# B&R Automation Studio project ComauRacer3demo (part 2)

### Config_3.mechanicalsystem - X20CP1586/mappMotion/6AxesRoboArmA/Config_3.mechanicalsystem
```
Element MechSys_6AxRobA (Type=mechanicalsystem)
  Type = 6AxesRoboarm
    Subtype = 6AxesRoboarmA
      Description = Standard
        Dimensions:
          TranslationFromBaseToQ1IsReadOnly = 0
          TranslationFromBaseToQ1:
            X = 0.0
            Y = 0.0
            Z = 0.0
          TranslationFromQ1ToQ2IsReadOnly = 0
          TranslationFromQ1ToQ2:
            X = 250.0
            Y = 0.0
            Z = 640.0
          TranslationFromQ2ToQ3IsReadOnly = 0
          TranslationFromQ2ToQ3:
            X = 0.0
            Y = 0.0
            Z = 630.0
          TranslationFromQ3ToQ4IsReadOnly = 0
          TranslationFromQ3ToQ4:
            X = 827.5
            Y = 0.0
            Z = 196.0
          TranslationFromQ4ToQ5IsReadOnly = 0
          TranslationFromQ4ToQ5:
            X = 0.0
          TranslationFromQ5ToQ6IsReadOnly = 0
          TranslationFromQ5ToQ6:
            X = 160.0
          TranslationFromQ6ToFlange:
            X = 0.0
            Y = 0.0
            Z = 0.0
        Offsets:
          JointAxisIsReadOnly = 0
          JointAxis[1] = 0.0
          JointAxis[2] = 0.0
          JointAxis[3] = 0.0
          JointAxis[4] = 0.0
          JointAxis[5] = 0.0
          JointAxis[6] = 0.0
        CountDirections:
          JointAxisIsReadOnly = 0
          JointAxis[1] = Standard
          JointAxis[2] = Standard
          JointAxis[3] = Standard
          JointAxis[4] = Standard
          JointAxis[5] = Standard
          JointAxis[6] = Standard
      CoordinatesNames = Default
        XCoordinateName = X
        YCoordinateName = Y
        ZCoordinateName = Z
        ACoordinateName = A
        BCoordinateName = B
        CCoordinateName = C
      WireFrameModel = Standard
        Q1ToQ2 = ConnectionLine
          Distance = 0.0
        Q2ToQ3 = ConnectionLine
          Distance = 0.0
        Q3ToQ4 = ConnectionLine
          Distance = 0.0
        Q4ToQ5 = ConnectionLine
          Distance = 0.0
        Q5ToQ6 = ConnectionLine
          Distance = 0.0
        Q6ToFlange = ConnectionLine
          Distance = 0.0
        FlangeToTcp = ConnectionLine
          Distance = 0.0
      DynamicModel = DynParTable
        TableRef
      InternalDynamicModel = NotUsed
      JointAxesPositionLimits:
        JointAxis[1] = UseAxisLimits
        JointAxis[2] = UseAxisLimits
        JointAxis[3] = UseAxisLimits
        JointAxis[4] = UseAxisLimits
        JointAxis[5] = UseAxisLimits
        JointAxis[6] = UseAxisLimits
```

## Logical view

Binary libraries used (declarations not repeated): operator, runtime, astime, AsIecCon, MpRobotics, McAxGroup, MpBase, McBase, CoTrace, AsZip, FileIO, sys_lib, McAcpAx, McAxis, MpAxis, McAcpPar, McPathGen, McProgInt, MpAudit 5.14.1, MpServer, MpAlarmX 5.14.1, MpUserX 5.14.1, MpFile 5.14.1, AsBrStr, MpRecipe 5.14.1

### Global.typ - Global data types
```iecst
TYPE
	R3ManualModeType : 	STRUCT  (*Manual mode type*)
		AxisButton : R3TCPAxisBtnType; (*Stores button states for global coordinate system*)
		JointButton : R3JointBtnType; (*Stores button states for axis coordinate system*)
		Velocity : REAL; (*Stores set velocity*)
		Acceleration : REAL; (*Stores set acceleration*)
		Deceleration : REAL; (*Stores set deceleration*)
		CoordinateSystem : UDINT; (*Stores selected coordinate system (0 - axis, 9 - global, 10 - tool) (no tool is set, so 9=10)*)
		Direction : DirectionEnum; (*Stores which direction should the axis be moved*)
	END_STRUCT;
	R3JointBtnType : 	STRUCT  (*Axes 1-6 select button*)
		Q1 : BOOL;
		Q2 : BOOL;
		Q3 : BOOL;
		Q4 : BOOL;
		Q5 : BOOL;
		Q6 : BOOL;
	END_STRUCT;
	R3TCPAxisBtnType : 	STRUCT  (*Global Coordinate System Select button*)
		X : BOOL;
		Y : BOOL;
		Z : BOOL;
		A : BOOL;
		B : BOOL;
		C : BOOL;
	END_STRUCT;
	DirectionEnum :
		(
		POSITIVE,
		NEGATIVE
		);
END_TYPE
```

### Global.var - Global variables
```iecst
VAR RETAIN
	gIsCalibrated : BOOL;
	gRacer3HomeRestorePos : ARRAY[0..5] OF McAcpAxRestorePosType; (*Permanent - stores home position, set in calibration process*)
	gRacer3ZeroPosition : ARRAY[0..5] OF LREAL; (*Position of axes saved after calibration*)
END_VAR
VAR
	gActiveContent : INT := 1;
END_VAR
```

### Package Logical/Libraries - Global libraries

### Library Logical/Libraries/RacerLib (IEC)

#### Types.typ - Exported data types
```iecst
TYPE
	R3AutomaticModeErrorEnum :
		(
		autoNO_ERROR := 0,
		autoLOAD_PROGRAM_ERROR := 1,
		autoUNLOAD_PROGRAM_ERROR := 2,
		autoEXECUTE_PROGRAM_ERROR := 3,
		autoPAUSE_ERROR := 4,
		autoCONTINUE_ERROR := 5,
		autoABORT_ERROR := 6
		);
	R3AutomaticModeCmds : 	STRUCT  (*Automatic mode commands*)
		LoadProgram : MC_BR_LoadProgram;
		ExecuteProgram : MC_BR_MoveProgram;
		UnloadProgram : MC_BR_UnloadProgram;
		PauseProgram : MC_GroupInterrupt;
		ContinueProgram : MC_GroupContinue;
		GroupStop : MC_GroupStop;
	END_STRUCT;
	R3AutomaticModeState :
		( (*Automatic mode state machine*)
		autoSTATE_WAIT := 1, (*waiting for instruction*)
		autoSTATE_LOAD := 2, (*loading program*)
		autoSTATE_UNLOAD := 3, (*Unloading program state*)
		autoSTATE_EXECUTE := 4, (*executing program*)
		autoSTATE_DONE := 5, (*execution done*)
		autoSTATE_PAUSE := 6, (*program paused*)
		autoSTATE_CONTINUE := 7, (*Continues paused program*)
		autoSTATE_ABORT := 8, (*Abort current program*)
		autoSTATE_ERROR := 0 (*error state*)
		);
	R3AutomaticModePara : 	STRUCT  (*Automatic mode parameters*)
		ProgramName : STRING[260]; (*Program name to load/execute*)
		Load : BOOL; (*Load a program*)
		Execute : BOOL; (*Executes a program*)
		Unload : BOOL; (*Unloads a program*)
		ErrorReset : BOOL; (*Resets errors*)
		Abort : BOOL; (*Aborts execution.*)
		UnloadAll : BOOL; (*tells the program to unload all programs from memory (used with Unload)*)
		Pause : BOOL; (*Pauses execution*)
		Continue : BOOL; (*Continues execution*)
		Continuous : BOOL; (*Defines whether the program will be called continuously*)
	END_STRUCT;
	R3AutomaticModeInfo : 	STRUCT
		CurrentState : R3AutomaticModeState; (*Current automode state*)
		Error : R3AutomaticModeErrorEnum;
		ErrorID : DINT;
		Paused : BOOL;
		IsError : BOOL; (*Only for visualisation.*)
	END_STRUCT;
	R3AutomaticModeType : 	STRUCT  (*Automatic mode main structure*)
		Parameters : R3AutomaticModePara;
		Info : R3AutomaticModeInfo;
		Cmds : R3AutomaticModeCmds;
	END_STRUCT;
	R3WorkspaceType : 	STRUCT  (*this allows workspace to be set during runtime.*)
		Para : McCfgAxGrpFeatWsmType := (ModalDataBehaviour:=(Type:=mcAGFMDB_USE_AX_GRP_SET));
		Cmd : MC_BR_ProcessConfig;
		Done : BOOL; (*indicates the FB has finished*)
	END_STRUCT;
	R3ManualModeType : 	STRUCT  (*Manual mode type*)
		AxisButton : R3AxisBtnType; (*Stores button states for select coordinate system*)
		CoordinateSystem : McCoordinateSystemEnum; (*Stores selected coordinate system (0 - axis, 9 - global, 10 - tool) (no tool is set, so 9=10)*)
		Direction : INT; (*Stores which direction should the axis be moved (1 - POSITIVE, -1 - NEGATIVE)*)
		JogVelocity : REAL := 20; (*Stores the velocity of axis*)
		PathLimits : McJogPathLimitsType; (*Stores set limits of acceleration and deceleration, velocity and jerk*)
		ActivateMove : BOOL; (*Enables or disables current move execution*)
		ExitManual : BOOL; (*Exits Manual Mode on True*)
	END_STRUCT;
	R3AxisBtnType : 	STRUCT  (*Global Coordinate System Select button*)
		Q1 : BOOL;
		Q2 : BOOL;
		Q3 : BOOL;
		Q4 : BOOL;
		Q5 : BOOL;
		Q6 : BOOL;
	END_STRUCT;
	R3DirectionEnum :
		( (*Currently unused*)
		POSITIVE := 1,
		NEGATIVE := -1
		);
	R3StateMachineEnum :
		(
		STATE_ERROR, (*Error state*)
		STATE_INIT, (*Initialisation state*)
		STATE_POWER_ON, (*Powering on state*)
		STATE_READY, (*Ready for commands*)
		STATE_MANUAL_CONTROL, (*Manual mode*)
		STATE_SEMI_AUTOMATIC, (*Semi automatic mode*)
		STATE_AUTOMATIC, (*Automatic mode (script execution)*)
		STATE_CALIBRATION, (*Calibration mode*)
		STATE_HOMING, (*Homing mode*)
		STATE_BRAKES (*This will read brakes' status.*)
		);
	R3CalibrationType : 	STRUCT
		CalibrationState : R3CalibrationStateEnum; (*State machine used to control Calibration behaviour*)
		CalibrationModePara : R3ManualModeType; (*same type used for manual mode (slightly different code handling)*)
		AxisCalibrated : ARRAY[0..5]OF BOOL := [6(0)]; (*Saves which axes have been calibrated (defaults to 0 upon creation)*)
		AxisSaveBtn : BOOL; (*Button to save current position as calibrated*)
		Axis5To6Para : R3Axis5To6Type; (*Stores axis 4 and 5 settings for axis 5 and 6 calibration*)
		SavedPositions : ARRAY[0..5]OF LREAL;
		InitHome : MC_BR_InitHome_AcpAx; (*Used to init home positions after each save*)
		InitHomePara : McAcpAxHomingParType; (*Homing parameters after each save*)
		AxesRef : ARRAY[0..5]OF UDINT; (*Axes reference.*)
	END_STRUCT;
	R3CalibrationStateEnum :
		(
		STATE_START,
		STATE_CALIBRATE_Q1,
		STATE_CALIBRATE_Q2,
		STATE_CALIBRATE_Q3,
		STATE_CALIBRATE_Q4,
		STATE_CALIBRATE_Q5,
		STATE_CALIBRATE_Q6,
		STATE_RESTORE_Q3_Q5
		);
	R3Axis5To6Type : 	STRUCT  (*Type for storing axis 3 and 5 settings for axes 5 and 6 calibration*)
		Axis3Moved : BOOL; (*Stores whether axis 3 has been moved in order to calibrate axes 5 and  6*)
		Axis5Moved : BOOL; (*Stores whether axis 5 has been moved in order to calibrate axis 6*)
		AxisMoveVelocity : REAL; (*Velocity of axis 3 and 5*)
		Axis3Angle : LREAL := -45.0; (*Angle of axis 3 to be set*)
		Axis5Angle : LREAL := -118.0; (*Angle of axis 5 to be set*)
		Axis5Return : BOOL; (*Flag to be set by a button to restore axis 3 and 5's positions after calibrating axis 6*)
		Axis35Restored : BOOL; (*Axis 3 and 5 have been restored to previous position*)
	END_STRUCT;
	R3SemiAutoEnumType :
		(
		INIT := 0,
		START := 1,
		UPDATE := 2,
		GO := 3,
		STATE_STOP := 5,
		STATE_PAUSE := 4
		);
	R3SemiAutoModeType : 	STRUCT
		AskedValue : R3AskedValueType; (*Stores given axis distance for relative move*)
		Flag : BOOL; (*Flag between READY and SEMIAUTO*)
		Mode : BOOL; (*Switches between relative and absolute modes, 1 for Relative, 0 for Absolute*)
		UpdatePending : BOOL; (*if UpdatePending then updates before starting move*)
		State : R3SemiAutoEnumType; (*state selector for state machine*)
		ModeForThisMove : BOOL; (*makes sure that switching mode in time of moving doesnt bugs out move*)
		CoordinateSystem : McCoordinateSystemEnum; (*Stores selected coordinate system (0 - axis, 9 - global, 10 - tool) (no tool is set, so 9=10)*)
		PathMode : BOOL; (*Switches between direct and linear path mode, 1 for linear , 0 for direct*)
		PathModeForThisMove : BOOL;
		ExitSemiAuto : BOOL;
		Pause : BOOL;
	END_STRUCT;
	ControlSelectEnum :
		(
		ManualJog := 1,
		SemiAutomatic := 2,
		Automatic := 3,
		None := 0
		);
	R3AskedValueType : 	STRUCT  (*for SemiAuto*)
		Velocity : REAL := 69;
		Acceleration : REAL := 100;
		Deceleration : REAL := 100;
		Jerk : REAL := 0;
		TCS : ARRAY[0..5]OF REAL := [420,420,420,69,69,69];
		ACS : ARRAY[0..5]OF REAL := [-69,69,69,69,-69,69];
	END_STRUCT;
	R3CalibrationMainType : 	STRUCT
		Info : CalibrationInfo; (*Information portion of calibration.*)
		Cmds : CalibrationCmds; (*Calibration commands*)
		Para : CalibrationParaType; (*Calibration parameters*)
	END_STRUCT;
	CalibrationParaType : 	STRUCT
		Parameters : R3CalibrationType;
		HomingParameters : McAcpAxHomingParType;
		FakeHomingModeEnum : ARRAY[0..14]OF McHomingModeEnum := [15(mcHOMING_DIRECT)];
		Positions : ARRAY[0..14]OF LREAL := [15(0.0)];
		HomingModeEnum : ARRAY[0..14]OF McHomingModeEnum := [15(mcHOMING_INIT)];
	END_STRUCT;
	CalibrationCmds : 	STRUCT
		Mode : R3CalibrationMode;
		InitHome : MC_BR_InitHome_AcpAx;
		GroupHome : MC_BR_GroupHome_15;
	END_STRUCT;
	CalibrationInfo : 	STRUCT
		CurrentState : OuterCalibrationState;
	END_STRUCT;
	OuterCalibrationState :
		(
		STATE_BEGIN,
		STATE_FAKE_HOME,
		STATE_MOVING,
		STATE_SAVING_POSITION,
		STATE_DONE
		);
	CommunicationType : 	STRUCT
		Power : BOOL := FALSE;
		Pause : BOOL := FALSE;
		Stop : BOOL := FALSE;
		ErrorReset : BOOL := FALSE;
		ModeSystem : BOOL := TRUE;
		PathSystem : BOOL := TRUE;
		changeModePending : USINT := 0; (*1-Manual       2-SemiManual      3-Auto 0-none*)
		NOTPathSystem : BOOL;
		NOTModeSystem : BOOL;
		CoordinateSystemManual : BOOL := FALSE;
		NOTCoordinateSystemSemiAuto : BOOL := FALSE;
		CoordinateSystemSemiAuto : BOOL := FALSE;
		NOTCoordinateSystem : BOOL;
		txt_State_out : WSTRING[80];
		AskedMaxVelocity : REAL; (*not needed*)
		AskedMaxAcc : REAL; (*not needed*)
		AskedMaxDeAcc : REAL; (*not needed*)
		AskedAutoJerk : REAL; (*not needed*)
		AskedAutoDeAcc : REAL; (*not needed*)
		AskedAutoAcc : REAL; (*not needed*)
		AskedAutoVelocity : REAL; (*not needed*)
		AskedManualVelocity : REAL; (*not needed*)
		UpdateSemiAutoVars : BOOL := FALSE;
		CalibBtn1To5 : BOOL := FALSE;
		CalibrationImage : STRING[80];
		TextManager : TextManagerType;
		RestoreAxis5 : BOOL := FALSE;
		CalibrateAgain : BOOL := FALSE;
		txt_State_out_front : STRING[80];
		BrakeOpen : BOOL; (*open the brakes*)
		BrakeClose : BOOL; (*close the brakes*)
		BrakeReadStatus : BOOL; (*read status of brakes*)
		BrakesSet : BOOL; (*This variable tells the program if brake parameters have been set.*)
		ToolOutput : BOOL; (*This variable enables tool control*)
		ReturnToZero : BOOL; (*This variable allows returning to zero position in manual mode.*)
		ResetHome : BOOL;
		WarmRestart : BOOL := FALSE;
		ReadWorkspace : BOOL;
	END_STRUCT;
	R3BrakeStateMachineEnum :
		(
		brakeREAD,
		brakeOPEN,
		brakeCLOSE,
		brakeDONE,
		brakeERROR
		);
	R3BrakeParaType : 	STRUCT
		BrakeCmd : McBrakeCmdEnum;
		Identifier : UDINT;
	END_STRUCT;
	R3BrakeCmdsType : 	STRUCT
		BrakeOperation : MC_BR_GroupBrakeOperation;
	END_STRUCT;
	R3BrakeInfoType : 	STRUCT
		BrakeStatus : ARRAY[1..2]OF McBrakeStatusEnum;
		Done : BOOL;
		State : R3BrakeStateMachineEnum;
		Error : BOOL;
	END_STRUCT;
	R3BrakeType : 	STRUCT
		Parameters : R3BrakeParaType;
		Info : R3BrakeInfoType;
		Cmds : R3BrakeCmdsType;
	END_STRUCT;
	R3KeyCheckType : 	STRUCT
		original_combo : ARRAY[0..4]OF USINT := [1,2,3,0,17];
		pending_combo : ARRAY[0..4]OF USINT;
		i : USINT := 0;
		temp_value : USINT;
		value_changed : BOOL := FALSE;
		event_achieved : BOOL := FALSE;
	END_STRUCT;
	TextManagerType : 	STRUCT
		CalibHelper : STRING[80];
	END_STRUCT;
END_TYPE
```

#### Constants.var - Exported constants
```iecst
VAR CONSTANT
	gAlarmXCore : USINT := 0;
END_VAR
```

#### RacerLib.fun - Exported functions and function blocks
```iecst
FUNCTION_BLOCK R3BrakeSet
	VAR_INPUT
		Axis1 : REFERENCE TO UDINT;
		Axis2 : REFERENCE TO UDINT;
		Axis3 : REFERENCE TO UDINT;
		Axis4 : REFERENCE TO UDINT;
		Axis5 : REFERENCE TO UDINT;
		Axis6 : REFERENCE TO UDINT;
	END_VAR
	VAR_OUTPUT
		Done : BOOL;
		Error : BOOL;
	END_VAR
	VAR
		BrakePara : McAcpAxBrakeParType;
		CurrentAxis : USINT := 1;
		BrakeSet : MC_BR_BrakeSetPar_AcpAx;
	END_VAR
END_FUNCTION_BLOCK

{REDUND_ERROR} FUNCTION_BLOCK R3ManualMode (*TODO: Add your comment here*) (*$GROUP=User,$CAT=User,$GROUPICON=User.png,$CATICON=User.png*)
	VAR_INPUT
		ManualModePara : R3ManualModeType;
	END_VAR
	VAR_IN_OUT
		RoboArm : MpRoboArm6Axis;
		RoboArmPara : MpRoboArm6AxisParType;
		MainState : R3StateMachineEnum;
		ControlSelector : ControlSelectEnum;
	END_VAR
	VAR
		j : USINT;
		JogVelocityActual : REAL;
	END_VAR
END_FUNCTION_BLOCK

{REDUND_ERROR} FUNCTION_BLOCK R3SemiAutoMode (*TODO: Add your comment here*) (*$GROUP=User,$CAT=User,$GROUPICON=User.png,$CATICON=User.png*)
	VAR_IN_OUT
		SemiAutoModePara : R3SemiAutoModeType;
		RoboArm : MpRoboArm6Axis;
		RoboArmPara : MpRoboArm6AxisParType;
		MainState : R3StateMachineEnum;
		ControlSelector : ControlSelectEnum;
	END_VAR
	VAR
		SemiAutoModePara_memory : R3SemiAutoModeType;
		WeNeedToGoBack : BOOL;
		IsPaused : BOOL;
	END_VAR
END_FUNCTION_BLOCK

{REDUND_UNREPLICABLE} FUNCTION_BLOCK R3CalibrationMode
	VAR_IN_OUT
		CalibrationPara : R3CalibrationType;
		RoboArm : MpRoboArm6Axis;
		RoboArmPara : MpRoboArm6AxisParType;
	END_VAR
	VAR
		JogVelocityActual : {REDUND_UNREPLICABLE} REAL;
		j : {REDUND_UNREPLICABLE} USINT;
	END_VAR
END_FUNCTION_BLOCK

{REDUND_ERROR} FUNCTION checkAxisLimits : BOOL (*returns TRUE if semi-automatic path is containted in axis limits, check is for relative positions*) (*$GROUP=User,$CAT=User,$GROUPICON=User.png,$CATICON=User.png*)
	VAR_INPUT
		Q1 : REAL;
		Q2 : REAL;
		Q3 : REAL;
		Q4 : REAL;
		Q5 : REAL;
		Q6 : REAL;
		Mode : BOOL; (*1 for relative, 0 for absolute*)
		RoboArm : MpRoboArm6Axis; (*needed for current axis position*)
	END_VAR
END_FUNCTION

{REDUND_ERROR} {REDUND_UNREPLICABLE} FUNCTION_BLOCK R3AutomaticMode (*TODO: Add your comment here*) (*$GROUP=User,$CAT=User,$GROUPICON=User.png,$CATICON=User.png*)
	VAR_INPUT
		AxesGroup : REFERENCE TO UDINT; (*AxesGroup to execute program on*)
	END_VAR
	VAR_IN_OUT
		AutoMode : R3AutomaticModeType; (*Main type variable*)
	END_VAR
	VAR
		UnloadMode : {REDUND_UNREPLICABLE} McUnloadProgramModeEnum; (*defines unload mode behaviour*)
	END_VAR
END_FUNCTION_BLOCK

{REDUND_ERROR} {REDUND_UNREPLICABLE} FUNCTION_BLOCK R3Workspace (*TODO: Add your comment here*) (*$GROUP=User,$CAT=User,$GROUPICON=User.png,$CATICON=User.png*)
	VAR_IN_OUT
		Para : R3WorkspaceType;
	END_VAR
END_FUNCTION_BLOCK
```

#### R3ManualMode.st
```iecst
(* TODO: Add your comment here *)
FUNCTION_BLOCK R3ManualMode

	IF ManualModePara.Direction = 1 THEN // set actual axis velocity based on which direction it's set to be moved
		JogVelocityActual := ManualModePara.JogVelocity;
	ELSIF ManualModePara.Direction = -1 THEN
		JogVelocityActual := -1 * ManualModePara.JogVelocity;
	ELSIF  ManualModePara.Direction = 0 THEN
		JogVelocityActual := 0;
	END_IF

	RoboArmPara.Jog.CoordSystem := ManualModePara.CoordinateSystem;
	RoboArmPara.Jog.PathLimits := ManualModePara.PathLimits;

	IF ManualModePara.ActivateMove THEN
		(* old Szymon's version
		IF ManualModePara.AxisButton.Q1 THEN // if a button is pressed, write corresponding velocity to the jog velocity array
			//IF RoboArmPara.Jog.Velocity[0] <> JogVelocityActual THEN // test if this fixes strange movement style
				RoboArmPara.Jog.Velocity[0] := JogVelocityActual;
			//END_IF
		ELSIF ManualModePara.AxisButton.Q2 THEN
			//IF RoboArmPara.Jog.Velocity[1] <> JogVelocityActual THEN
				RoboArmPara.Jog.Velocity[1] := JogVelocityActual;
			//END_IF
		ELSIF ManualModePara.AxisButton.Q3 THEN
			RoboArmPara.Jog.Velocity[2] := JogVelocityActual;

		ELSIF ManualModePara.AxisButton.Q4 THEN
			RoboArmPara.Jog.Velocity[3] := JogVelocityActual;

		ELSIF ManualModePara.AxisButton.Q5 THEN
			RoboArmPara.Jog.Velocity[4] := JogVelocityActual;

		ELSIF ManualModePara.AxisButton.Q6 THEN
			RoboArmPara.Jog.Velocity[5] := JogVelocityActual;

		ELSE //if no buttons are pressed reset jog velocity array

			FOR j := 0 TO 5 BY 1 DO //set every jog velocity to 0
				RoboArmPara.Jog.Velocity[j] := 0.0;
			END_FOR;
		END_IF
		*)

		IF ManualModePara.AxisButton.Q1 THEN
			RoboArmPara.Jog.Velocity[0] := JogVelocityActual;
		ELSE
			RoboArmPara.Jog.Velocity[0] := 0;
		END_IF

		IF ManualModePara.AxisButton.Q2 THEN
			RoboArmPara.Jog.Velocity[1] := JogVelocityActual;
		ELSE
			RoboArmPara.Jog.Velocity[1] := 0;
		END_IF

		IF ManualModePara.AxisButton.Q3 THEN
			RoboArmPara.Jog.Velocity[2] := JogVelocityActual;
		ELSE
			RoboArmPara.Jog.Velocity[2] := 0;
		END_IF

		IF ManualModePara.AxisButton.Q4 THEN
			RoboArmPara.Jog.Velocity[3] := JogVelocityActual;
		ELSE
			RoboArmPara.Jog.Velocity[3] := 0;
		END_IF

		IF ManualModePara.AxisButton.Q5 THEN
			RoboArmPara.Jog.Velocity[4] := JogVelocityActual;
		ELSE
			RoboArmPara.Jog.Velocity[4] := 0;
		END_IF

		IF ManualModePara.AxisButton.Q6 THEN
			RoboArmPara.Jog.Velocity[5] := JogVelocityActual;
		ELSE
			RoboArmPara.Jog.Velocity[5] := 0;
		END_IF
		IF RoboArm.Jog <> TRUE THEN
			RoboArm.Jog := TRUE;
		END_IF
	ELSE
		RoboArm.Jog := FALSE;
	END_IF

	IF ManualModePara.ExitManual THEN
		//clean up
		ManualModePara.Direction:=0;
		JogVelocityActual:=0;
		FOR j := 0 TO 5 BY 1 DO //set every jog velocity to 0
				RoboArmPara.Jog.Velocity[j] := 0;
		END_FOR;
		ManualModePara.ActivateMove:=FALSE;
		RoboArm.Jog:=FALSE;
		//go out
		ManualModePara.ExitManual := FALSE;
	END_IF

END_FUNCTION_BLOCK
```

#### R3SemiAutoMode.st
```iecst
FUNCTION_BLOCK R3SemiAutoMode

	IF SemiAutoModePara.ExitSemiAuto THEN
		SemiAutoModePara.State := STATE_STOP;
	END_IF

	(*
	IF SemiAutoModePara.Pause THEN
		SemiAutoModePara_memory := SemiAutoModePara;
		RoboArm.MoveDirect:=FALSE;
		RoboArm.MoveLinear:=FALSE;
		SemiAutoModePara.Flag:=FALSE;
	END_IF
	*)
	CASE SemiAutoModePara.State OF
		INIT:
			IF SemiAutoModePara.UpdatePending THEN
				SemiAutoModePara.State := UPDATE;
			ELSE
				SemiAutoModePara.State := START;
			END_IF

			//TODO CHECK AXIS LIMITS AND SINGULAR POINT AND SEND ERROR (ALARM) AND AVOID MOVING
			//IF checkAxisLimits(Q1:=SemiAutoModePara.AskedValue.Q0,Q2:=SemiAutoModePara.AskedValue.Q1,Q3:=SemiAutoModePara.AskedValue.Q2,Q4:=SemiAutoModePara.AskedValue.Q3,Q5:=SemiAutoModePara.AskedValue.Q4,Q6:=SemiAutoModePara.AskedValue.Q5,Mode := SemiAutoModePara.ModeForThisMove, RoboArm:=RoboArm) THEN
			// send alarm out of bounds
			//MpAlarmXSet(gAlarmXCore, 'OutOfLimits');
			//END_IF

			// check for singular point and send alarm

		UPDATE:

			RoboArmPara.CoordSystem := SemiAutoModePara.CoordinateSystem;

			RoboArmPara.Velocity := SemiAutoModePara.AskedValue.Velocity;
			RoboArmPara.Acceleration := SemiAutoModePara.AskedValue.Acceleration;
			RoboArmPara.Deceleration := SemiAutoModePara.AskedValue.Deceleration;
			RoboArmPara.Jerk := SemiAutoModePara.AskedValue.Jerk;

			SemiAutoModePara.ModeForThisMove:=SemiAutoModePara.Mode;
			SemiAutoModePara.PathModeForThisMove:=SemiAutoModePara.PathMode;

			IF SemiAutoModePara.CoordinateSystem = 0 THEN // ACS
				IF SemiAutoModePara.ModeForThisMove THEN //relative
					RoboArmPara.Distance[0] := SemiAutoModePara.AskedValue.ACS[0];
					RoboArmPara.Distance[1] := SemiAutoModePara.AskedValue.ACS[1];
					RoboArmPara.Distance[2] := SemiAutoModePara.AskedValue.ACS[2];
					RoboArmPara.Distance[3] := SemiAutoModePara.AskedValue.ACS[3];
					RoboArmPara.Distance[4] := SemiAutoModePara.AskedValue.ACS[4];
					RoboArmPara.Distance[5] := SemiAutoModePara.AskedValue.ACS[5];
				ELSE //absolute
					RoboArmPara.Position[0] := SemiAutoModePara.AskedValue.ACS[0];
					RoboArmPara.Position[1] := SemiAutoModePara.AskedValue.ACS[1];
					RoboArmPara.Position[2] := SemiAutoModePara.AskedValue.ACS[2];
					RoboArmPara.Position[3] := SemiAutoModePara.AskedValue.ACS[3];
					RoboArmPara.Position[4] := SemiAutoModePara.AskedValue.ACS[4];
					RoboArmPara.Position[5] := SemiAutoModePara.AskedValue.ACS[5];
				END_IF
			ELSIF SemiAutoModePara.CoordinateSystem = 9 THEN // TCS
				IF SemiAutoModePara.ModeForThisMove THEN //relative
					RoboArmPara.Distance[0] := SemiAutoModePara.AskedValue.TCS[0];
					RoboArmPara.Distance[1] := SemiAutoModePara.AskedValue.TCS[1];
					RoboArmPara.Distance[2] := SemiAutoModePara.AskedValue.TCS[2];
					RoboArmPara.Distance[3] := SemiAutoModePara.AskedValue.TCS[3];
					RoboArmPara.Distance[4] := SemiAutoModePara.AskedValue.TCS[4];
					RoboArmPara.Distance[5] := SemiAutoModePara.AskedValue.TCS[5];
				ELSE //absolute
					RoboArmPara.Position[0] := SemiAutoModePara.AskedValue.TCS[0];
					RoboArmPara.Position[1] := SemiAutoModePara.AskedValue.TCS[1];
					RoboArmPara.Position[2] := SemiAutoModePara.AskedValue.TCS[2];
					RoboArmPara.Position[3] := SemiAutoModePara.AskedValue.TCS[3];
					RoboArmPara.Position[4] := SemiAutoModePara.AskedValue.TCS[4];
					RoboArmPara.Position[5] := SemiAutoModePara.AskedValue.TCS[5];
				END_IF
			END_IF

			IF SemiAutoModePara.Mode THEN
				RoboArmPara.ManualMoveType := 1;
			ELSE
				RoboArmPara.ManualMoveType := 0;
			END_IF
			RoboArm.Update:= TRUE;
			IF RoboArm.UpdateDone THEN
				RoboArm.Update:=FALSE;
				SemiAutoModePara.UpdatePending:=FALSE;
				SemiAutoModePara.State := START;
				WeNeedToGoBack:=FALSE;
			END_IF
		START:
			IF SemiAutoModePara.UpdatePending THEN
				SemiAutoModePara.State:=UPDATE;
				WeNeedToGoBack := TRUE;
			END_IF
			IF SemiAutoModePara.Flag AND NOT WeNeedToGoBack THEN
				IF SemiAutoModePara.PathModeForThisMove THEN
					RoboArm.MoveLinear:=TRUE;
				ELSE
					RoboArm.MoveDirect:=TRUE;
				END_IF
				SemiAutoModePara.State:=GO;
			END_IF
		GO:
			IF NOT SemiAutoModePara.Flag THEN
				SemiAutoModePara.State:=STATE_STOP;
			END_IF
			IF RoboArm.MoveDone THEN
				IF SemiAutoModePara.PathModeForThisMove THEN
					RoboArm.MoveLinear:=FALSE;
				ELSE
					RoboArm.MoveDirect:=FALSE;
				END_IF
				SemiAutoModePara.State:=INIT;
				SemiAutoModePara.Flag:=FALSE;
				MainState := STATE_READY;
			END_IF
		STATE_STOP:
			RoboArm.MoveDirect:=FALSE;
			RoboArm.MoveLinear:=FALSE;
			SemiAutoModePara.Flag:=FALSE;
			SemiAutoModePara.State:=INIT;
			SemiAutoModePara.ExitSemiAuto:=FALSE;
		STATE_PAUSE:
			//TODO count movement deegrees in relative and substract so unpause in relative mode "continues"

	END_CASE
END_FUNCTION_BLOCK
```

#### R3CalibrationMode.st
```iecst
(* TODO: Add your comment here
ActivateMove and AxisSaveBtn are assumed momentary.
not resetting AxisSaveBtn and switching AxisButton will result in immediate AxisCalibrated[i] := TRUE!
not resetting ActivateMove might result in damage to physical system! *)
FUNCTION_BLOCK R3CalibrationMode
	IF CalibrationPara.InitHome.Done OR NOT CalibrationPara.InitHome.Busy OR CalibrationPara.InitHome.Error THEN
		CalibrationPara.InitHome(Execute := FALSE);
	END_IF

	CalibrationPara.InitHomePara.Position := 0.0; //this is non-zero only for Axis 3
	CalibrationPara.InitHomePara.HomingMode := mcHOMING_DIRECT; //this saves current position as value 'Position'
	IF CalibrationPara.InitHome.Done THEN
		CalibrationPara.InitHome(Execute := FALSE);
	END_IF

	IF CalibrationPara.CalibrationModePara.Direction = 1 THEN // set actual axis velocity based on which direction it's set to be moved

		JogVelocityActual := CalibrationPara.CalibrationModePara.JogVelocity;

	ELSIF CalibrationPara.CalibrationModePara.Direction = -1 THEN

		JogVelocityActual := -1 * CalibrationPara.CalibrationModePara.JogVelocity;

	END_IF

	CASE CalibrationPara.CalibrationState OF
		STATE_START:
			CalibrationPara.AxisSaveBtn := FALSE; //reset button status in case someone clicks when axis isn't ready
			IF RoboArm.MoveDirect THEN
				RoboArm.MoveDirect := FALSE;
			END_IF

			RoboArmPara.Jog.CoordSystem := CalibrationPara.CalibrationModePara.CoordinateSystem;
			RoboArmPara.Jog.PathLimits := CalibrationPara.CalibrationModePara.PathLimits;

			IF NOT CalibrationPara.CalibrationModePara.ActivateMove THEN //disable jog if "Move" flag isn't set
				RoboArm.Jog := FALSE;
				FOR j := 0 TO 5 BY 1 DO //set every jog velocity to 0
					RoboArmPara.Jog.Velocity[j] := 0.0;
				END_FOR;
			END_IF

			IF CalibrationPara.AxisSaveBtn THEN //if AxisSaveBtn flag is set, reset it
				CalibrationPara.AxisSaveBtn := FALSE;
			END_IF

			IF CalibrationPara.CalibrationModePara.AxisButton.Q1 THEN // if a button is pressed, write corresponding velocity to the jog velocity array
				CalibrationPara.CalibrationState := STATE_CALIBRATE_Q1;

			ELSIF CalibrationPara.CalibrationModePara.AxisButton.Q2 THEN
				CalibrationPara.CalibrationState := STATE_CALIBRATE_Q2;

			ELSIF CalibrationPara.CalibrationModePara.AxisButton.Q3 THEN
				CalibrationPara.CalibrationState := STATE_CALIBRATE_Q3;

			ELSIF CalibrationPara.CalibrationModePara.AxisButton.Q4 THEN
				CalibrationPara.CalibrationState := STATE_CALIBRATE_Q4;

			ELSIF CalibrationPara.CalibrationModePara.AxisButton.Q5 THEN
				CalibrationPara.CalibrationState := STATE_CALIBRATE_Q5;

			ELSIF CalibrationPara.CalibrationModePara.AxisButton.Q6 THEN //don't permit axis 6 calibration until all the others are calibrated!
				CalibrationPara.CalibrationState := STATE_CALIBRATE_Q6;
			END_IF

			IF CalibrationPara.Axis5To6Para.Axis5Return AND CalibrationPara.AxisCalibrated[5] AND NOT CalibrationPara.Axis5To6Para.Axis35Restored AND CalibrationPara.Axis5To6Para.Axis5Moved AND CalibrationPara.Axis5To6Para.Axis3Moved THEN
				//only allow this if axis 6 has been calibrated (Show button in HMI)
				CalibrationPara.CalibrationState := STATE_RESTORE_Q3_Q5;
			END_IF

		STATE_CALIBRATE_Q1:
			RoboArmPara.Jog.Velocity[0] := JogVelocityActual; //write jog velocity to robot

			IF CalibrationPara.CalibrationModePara.ActivateMove THEN //enable jog only if ActivateMove flag is set
				RoboArm.Jog := TRUE;
			ELSE
				RoboArm.Jog := FALSE;
			END_IF

			IF CalibrationPara.AxisSaveBtn THEN //set Calibrated flag for given axis if AxisSaveBtn flag is set
				CalibrationPara.AxisCalibrated[0] := TRUE;
				CalibrationPara.InitHome(Axis := (*ADR*)(CalibrationPara.AxesRef[0]), Execute := TRUE, HomingParameters := CalibrationPara.InitHomePara);
				CalibrationPara.SavedPositions[0] := CalibrationPara.InitHomePara.Position;
				RoboArm.Jog := FALSE;
				CalibrationPara.AxisSaveBtn := FALSE;
			END_IF

			IF NOT CalibrationPara.CalibrationModePara.AxisButton.Q1 THEN //go back if button is released
				CalibrationPara.CalibrationState := STATE_START;
			END_IF

		STATE_CALIBRATE_Q2:
			RoboArmPara.Jog.Velocity[1] := JogVelocityActual;

			IF CalibrationPara.CalibrationModePara.ActivateMove THEN //enable jog only if ActivateMove flag is set
				RoboArm.Jog := TRUE;
			ELSE
				RoboArm.Jog := FALSE;
			END_IF

			IF CalibrationPara.AxisSaveBtn THEN //set Calibrated flag for given axis if AxisSaveBtn flag is set
				CalibrationPara.AxisCalibrated[1] := TRUE;
				CalibrationPara.InitHome(Axis := (*ADR*)(CalibrationPara.AxesRef[1]), Execute := TRUE, HomingParameters := CalibrationPara.InitHomePara);
				CalibrationPara.SavedPositions[1] := CalibrationPara.InitHomePara.Position;
				RoboArm.Jog := FALSE;
				CalibrationPara.AxisSaveBtn := FALSE;
			END_IF

			IF NOT CalibrationPara.CalibrationModePara.AxisButton.Q2 THEN
				CalibrationPara.CalibrationState := STATE_START;
			END_IF

		STATE_CALIBRATE_Q3:
			RoboArmPara.Jog.Velocity[2] := JogVelocityActual;

			IF CalibrationPara.CalibrationModePara.ActivateMove THEN //enable jog only if ActivateMove flag is set
				RoboArm.Jog := TRUE;
			ELSE
				RoboArm.Jog := FALSE;
			END_IF

			IF CalibrationPara.AxisSaveBtn THEN //set Calibrated flag for given axis if AxisSaveBtn flag is set
				CalibrationPara.AxisCalibrated[2] := TRUE;
				CalibrationPara.InitHomePara.Position := -90.0;
				CalibrationPara.InitHome(Axis := (*ADR*)(CalibrationPara.AxesRef[2]), Execute := TRUE, HomingParameters := CalibrationPara.InitHomePara);
				CalibrationPara.SavedPositions[2] := CalibrationPara.InitHomePara.Position;
				RoboArm.Jog := FALSE;
				CalibrationPara.AxisSaveBtn := FALSE;
			END_IF

			IF NOT CalibrationPara.CalibrationModePara.AxisButton.Q3 THEN
				CalibrationPara.CalibrationState := STATE_START;
			END_IF

		STATE_CALIBRATE_Q4:
			RoboArmPara.Jog.Velocity[3] := JogVelocityActual;

			IF CalibrationPara.CalibrationModePara.ActivateMove THEN //enable jog only if ActivateMove flag is set
				RoboArm.Jog := TRUE;
			ELSE
				RoboArm.Jog := FALSE;
			END_IF

			IF CalibrationPara.AxisSaveBtn THEN //set Calibrated flag for given axis if AxisSaveBtn flag is set
				CalibrationPara.AxisCalibrated[3] := TRUE;
				CalibrationPara.InitHome(Axis := (*ADR*)(CalibrationPara.AxesRef[3]), Execute := TRUE, HomingParameters := CalibrationPara.InitHomePara);
				CalibrationPara.SavedPositions[3] := CalibrationPara.InitHomePara.Position;
				RoboArm.Jog := FALSE;
				CalibrationPara.AxisSaveBtn := FALSE;
			END_IF

			IF NOT CalibrationPara.CalibrationModePara.AxisButton.Q4 THEN
				CalibrationPara.CalibrationState := STATE_START;
			END_IF

		STATE_CALIBRATE_Q5:
			IF CalibrationPara.AxisCalibrated[0] AND CalibrationPara.AxisCalibrated[1] AND CalibrationPara.AxisCalibrated[2] AND CalibrationPara.AxisCalibrated[3] THEN //if axes 1-4 have been calibrated
				(*one-time execution of relative movement of axis 3 by -45 degrees*)
				IF NOT CalibrationPara.Axis5To6Para.Axis3Moved AND NOT RoboArm.MoveActive AND NOT RoboArm.MoveDirect THEN

					FOR j := 0 TO 5 BY 1 DO //set every distance to 0
						RoboArmPara.Distance[j] := 0.0;
					END_FOR;

					RoboArmPara.Distance[2] := CalibrationPara.Axis5To6Para.Axis3Angle; //axis 3 may be moved this amount in order to make calibrating axis 5 and 6 easier (default -45)
					RoboArmPara.Velocity := CalibrationPara.Axis5To6Para.AxisMoveVelocity; // use a low velocity for this (just to be safe)
					RoboArmPara.ManualMoveType := mcMOVE_RELATIVE; //select relative movement (to restore position after calibrating axis 6)
					RoboArmPara.CoordSystem := 0; // select ACS for moving
					RoboArm.MoveDirect := TRUE; //execute movement

				ELSIF RoboArm.MoveDone AND RoboArm.MoveDirect THEN //if move has been executed

					RoboArm.MoveDirect := FALSE; //reset move flag
					CalibrationPara.Axis5To6Para.Axis3Moved := TRUE; //set flag to let the program know axis 5 has been moved to correct position

				ELSIF CalibrationPara.Axis5To6Para.Axis3Moved THEN //actual calibration

					RoboArmPara.Jog.Velocity[4] := JogVelocityActual;

					IF CalibrationPara.CalibrationModePara.ActivateMove THEN //enable jog only if ActivateMove flag is set
						RoboArm.Jog := TRUE;
					ELSE
						RoboArm.Jog := FALSE;
					END_IF

					IF CalibrationPara.AxisSaveBtn THEN //set Calibrated flag for given axis if AxisSaveBtn flag is set
						CalibrationPara.AxisCalibrated[4] := TRUE;
						CalibrationPara.InitHome(Axis := (*ADR*)(CalibrationPara.AxesRef[4]), Execute := TRUE, HomingParameters := CalibrationPara.InitHomePara);
						CalibrationPara.SavedPositions[4] := CalibrationPara.InitHomePara.Position;
						RoboArm.Jog := FALSE;
						CalibrationPara.AxisSaveBtn := FALSE;
					END_IF

				END_IF

			END_IF

			IF NOT CalibrationPara.CalibrationModePara.AxisButton.Q5 THEN
				CalibrationPara.CalibrationState := STATE_START;
			END_IF

		STATE_CALIBRATE_Q6:
			(* if all previous axes have been calibrated and set in place *)
			IF CalibrationPara.AxisCalibrated[0] AND CalibrationPara.AxisCalibrated[1] AND CalibrationPara.AxisCalibrated[2] AND CalibrationPara.AxisCalibrated[3] AND CalibrationPara.AxisCalibrated[4] THEN
				(*one-time execution of relative movement of axis 5 by -118 degrees*)
				IF NOT CalibrationPara.Axis5To6Para.Axis5Moved AND NOT RoboArm.MoveActive AND NOT RoboArm.MoveDirect THEN

					FOR j := 0 TO 5 BY 1 DO //set every distance to 0
						RoboArmPara.Distance[j] := 0.0;
					END_FOR;

					RoboArmPara.Distance[4] := CalibrationPara.Axis5To6Para.Axis5Angle; //axis 5 has to be moved this amount in order to calibrate axis 6 (see page 100 of _lb-rc-RACER3-STM_en) (default -118.0)
					//axis 3 is assumed to have been moved in order to make calibrating axis 6 easier (default -45)
					RoboArmPara.Velocity := CalibrationPara.Axis5To6Para.AxisMoveVelocity; // use a low velocity for this (just to be safe)
					RoboArmPara.ManualMoveType := mcMOVE_RELATIVE; //select relative movement (to restore position after calibrating axis 6)
					RoboArmPara.CoordSystem := 0; // select ACS for moving
					RoboArm.MoveDirect := TRUE; //execute movement

				ELSIF RoboArm.MoveDone AND RoboArm.MoveDirect THEN //if move has been executed

					RoboArm.MoveDirect := FALSE; //reset move flag
					CalibrationPara.Axis5To6Para.Axis5Moved := TRUE; //set flag to let the program know axis 5 has been moved to correct position

				ELSIF CalibrationPara.Axis5To6Para.Axis5Moved THEN //actual calibration

					RoboArmPara.Jog.Velocity[5] := JogVelocityActual;

					IF CalibrationPara.CalibrationModePara.ActivateMove THEN //enable jog only if ActivateMove flag is set (momentary switch in HMI)
						RoboArm.Jog := TRUE;
					ELSE
						RoboArm.Jog := FALSE;
					END_IF

					IF CalibrationPara.AxisSaveBtn THEN //set Calibrated flag for given axis if AxisSaveBtn flag is set
						CalibrationPara.AxisCalibrated[5] := TRUE;
						CalibrationPara.InitHome(Axis := (*ADR*)(CalibrationPara.AxesRef[5]), Execute := TRUE, HomingParameters := CalibrationPara.InitHomePara);
						CalibrationPara.SavedPositions[5] := CalibrationPara.InitHomePara.Position;
						RoboArm.Jog := FALSE;
						CalibrationPara.AxisSaveBtn := FALSE;
					END_IF

				END_IF

			END_IF

			IF NOT CalibrationPara.CalibrationModePara.AxisButton.Q6 THEN
				CalibrationPara.CalibrationState := STATE_START;
			END_IF

		STATE_RESTORE_Q3_Q5:

			IF CalibrationPara.Axis5To6Para.Axis5Moved AND CalibrationPara.Axis5To6Para.Axis3Moved AND NOT RoboArm.MoveActive AND NOT RoboArm.MoveDirect THEN

				FOR j := 0 TO 5 BY 1 DO //set every distance to 0
					RoboArmPara.Distance[j] := 0.0;
				END_FOR;

				RoboArmPara.Distance[4] := -1 * CalibrationPara.Axis5To6Para.Axis5Angle; // simply move axis 5 by negative of what it was moved before (see page 100 of _lb-rc-RACER3-STM_en)
				RoboArmPara.Distance[2] := -1 * CalibrationPara.Axis5To6Para.Axis3Angle; //reverse the move done previously
				RoboArmPara.Velocity := CalibrationPara.Axis5To6Para.AxisMoveVelocity; // use a slow velocity for this (just to be safe)
				RoboArmPara.ManualMoveType := mcMOVE_RELATIVE; //select relative movement (to restore position after calibrating axis 6)
				RoboArmPara.CoordSystem := 0; // select ACS for moving
				RoboArm.MoveDirect := TRUE; //execute movement

			ELSIF RoboArm.MoveDone AND RoboArm.MoveDirect THEN //if move has been executed

				RoboArm.MoveDirect := FALSE; //reset move flag
				CalibrationPara.Axis5To6Para.Axis3Moved := FALSE;
				CalibrationPara.Axis5To6Para.Axis5Moved := FALSE; //set flag to let the program know axis 5 has been moved to correct position
				CalibrationPara.Axis5To6Para.Axis35Restored := TRUE;

			END_IF

			IF CalibrationPara.Axis5To6Para.Axis35Restored THEN
				CalibrationPara.Axis5To6Para.Axis5Return := FALSE;
				CalibrationPara.CalibrationState := STATE_START;
			END_IF

	END_CASE

END_FUNCTION_BLOCK
```

#### checkAxisLimits.st
```iecst
(* returns TRUE if semi-automatic path is containted in axis limits, check is for relative positions *)
FUNCTION checkAxisLimits
	// Q1 -170 170
	// Q2 -95 135
	// Q3 -155 90
	// Q4 -200 200
	// Q5 -125 125
	// Q6 -270 270
	checkAxisLimits:=TRUE;
	IF Mode THEN
	//relative
		IF RoboArm.Info.JointAxisPosition[0] + Q1 < -170 OR RoboArm.Info.JointAxisPosition[0] + Q1 > 170 THEN
			checkAxisLimits := FALSE;
		END_IF
		IF RoboArm.Info.JointAxisPosition[1] + Q2 < -95 OR RoboArm.Info.JointAxisPosition[1] + Q2 > 135 THEN
			checkAxisLimits := FALSE;
		END_IF
		IF RoboArm.Info.JointAxisPosition[2] + Q3 < -155 OR RoboArm.Info.JointAxisPosition[2] + Q3 > 90 THEN
			checkAxisLimits := FALSE;
		END_IF
		IF RoboArm.Info.JointAxisPosition[3] + Q4 < -200 OR RoboArm.Info.JointAxisPosition[3] + Q4 > 200 THEN
			checkAxisLimits := FALSE;
		END_IF
		IF RoboArm.Info.JointAxisPosition[4] + Q5 < -125 OR RoboArm.Info.JointAxisPosition[4] + Q5 > 125 THEN
			checkAxisLimits := FALSE;
		END_IF
		IF RoboArm.Info.JointAxisPosition[5] + Q6 < -270 OR RoboArm.Info.JointAxisPosition[5] + Q6 > 270 THEN
			checkAxisLimits := FALSE;
		END_IF
	ELSE
	//absolute
		IF Q1 < -170 OR  Q1 > 170 THEN
			checkAxisLimits := FALSE;
		END_IF
		IF Q2 < -95 OR Q2 > 135 THEN
			checkAxisLimits := FALSE;
		END_IF
		IF Q3 < -155 OR Q3 > 90 THEN
			checkAxisLimits := FALSE;
		END_IF
		IF Q4 < -200 OR Q4 > 200 THEN
			checkAxisLimits := FALSE;
		END_IF
		IF Q5 < -125 OR Q5 > 125 THEN
			checkAxisLimits := FALSE;
		END_IF
		IF Q6 < -270 OR Q6 > 270 THEN
			checkAxisLimits := FALSE;
		END_IF
	END_IF
END_FUNCTION
```

#### R3AutomaticMode.st
```iecst
(* TODO: Add your comment here *)
FUNCTION_BLOCK R3AutomaticMode

	IF AutoMode.Parameters.Abort THEN
		//aborts execution
		AutoMode.Info.CurrentState := autoSTATE_ABORT;
	ELSIF AutoMode.Parameters.Pause AND NOT AutoMode.Info.Paused THEN
		//pauses execution
		AutoMode.Info.CurrentState := autoSTATE_PAUSE;
	END_IF

	CASE AutoMode.Info.CurrentState OF
		autoSTATE_WAIT:
			IF NOT AutoMode.Info.Paused THEN
				AutoMode.Cmds.ExecuteProgram(AxesGroup := ADR(AxesGroup), Execute := FALSE);
				AutoMode.Cmds.UnloadProgram(AxesGroup := ADR(AxesGroup), Execute := FALSE);
				AutoMode.Cmds.LoadProgram(AxesGroup := ADR(AxesGroup), Execute := FALSE);

				AutoMode.Info.Error := autoNO_ERROR; //reset error status in case it didn't reset. also useful for first-time execution
				AutoMode.Info.ErrorID := 0;
				AutoMode.Info.IsError := FALSE;

				IF AutoMode.Parameters.Load THEN //if "Load" is set, reset others (only one button can be pressed at a time, with priority to whichever was first)

					AutoMode.Parameters.Execute := FALSE;
					AutoMode.Parameters.Unload := FALSE;
					AutoMode.Info.CurrentState := autoSTATE_LOAD;

				ELSIF AutoMode.Parameters.Execute THEN

					AutoMode.Parameters.Load := FALSE;
					AutoMode.Parameters.Unload := FALSE;
					AutoMode.Info.CurrentState := autoSTATE_EXECUTE;

				ELSIF AutoMode.Parameters.Unload THEN

					AutoMode.Parameters.Load := FALSE;
					AutoMode.Parameters.Execute := FALSE;
					AutoMode.Info.CurrentState := autoSTATE_UNLOAD;

				END_IF
			ELSIF AutoMode.Parameters.Continue THEN
				AutoMode.Info.CurrentState := autoSTATE_CONTINUE;
			END_IF

		autoSTATE_LOAD: //this state loads a program specified in "ProgramName"

			AutoMode.Cmds.LoadProgram(AxesGroup := ADR(AxesGroup), Execute := TRUE, Name := AutoMode.Parameters.ProgramName, Mode := mcLOADPRG_PROGRAM);

			IF AutoMode.Cmds.LoadProgram.Done THEN
				AutoMode.Info.CurrentState := autoSTATE_DONE;
				AutoMode.Parameters.Load := FALSE;
			ELSIF AutoMode.Cmds.LoadProgram.Error THEN
				AutoMode.Info.IsError := TRUE;
				AutoMode.Info.ErrorID := AutoMode.Cmds.LoadProgram.ErrorID;
				AutoMode.Info.Error := autoLOAD_PROGRAM_ERROR;
				AutoMode.Parameters.Load := FALSE;
				AutoMode.Info.CurrentState := autoSTATE_ERROR;
			END_IF

		autoSTATE_UNLOAD: //this state unloads a program specified in "ProgramName" OR all programs (UnloadAll = true) from memory

			IF AutoMode.Parameters.UnloadAll THEN
				UnloadMode := mcUNLOADPRG_ALL;
			ELSE
				UnloadMode := mcUNLOADPRG_PROGRAM;
			END_IF

			AutoMode.Cmds.UnloadProgram(AxesGroup := ADR(AxesGroup), Execute := TRUE, Name := AutoMode.Parameters.ProgramName, Mode := UnloadMode);

			IF AutoMode.Cmds.UnloadProgram.Done THEN
				AutoMode.Info.CurrentState := autoSTATE_DONE;
				AutoMode.Parameters.Unload := FALSE;
			ELSIF AutoMode.Cmds.UnloadProgram.Error THEN
				AutoMode.Info.IsError := TRUE;
				AutoMode.Info.ErrorID := AutoMode.Cmds.UnloadProgram.ErrorID;
				AutoMode.Info.Error := autoUNLOAD_PROGRAM_ERROR;
				AutoMode.Parameters.Unload := FALSE;
				AutoMode.Info.CurrentState := autoSTATE_ERROR;
			END_IF

		autoSTATE_EXECUTE: //this state executes a program specified in "ProgramName", if program isn't loaded it will automagically load it

			AutoMode.Cmds.ExecuteProgram(AxesGroup := ADR(AxesGroup), Execute := TRUE, Name := AutoMode.Parameters.ProgramName);

			IF AutoMode.Cmds.ExecuteProgram.Done AND NOT AutoMode.Parameters.Execute THEN //if "Execute" was reset during program execution, disable Continuous. (user pressed the button again)
				AutoMode.Parameters.Continuous := FALSE;
				AutoMode.Info.CurrentState := autoSTATE_DONE;

			ELSIF AutoMode.Cmds.ExecuteProgram.Done AND AutoMode.Parameters.Execute THEN //if Execute is set after program execution, simply go to the Done state and handle Continuous there.
				AutoMode.Parameters.Execute := FALSE;
				AutoMode.Info.CurrentState := autoSTATE_DONE;

			ELSIF AutoMode.Cmds.ExecuteProgram.Error THEN //save error ID and go to error state
				AutoMode.Info.IsError := TRUE;
				AutoMode.Info.ErrorID := AutoMode.Cmds.ExecuteProgram.ErrorID;
				AutoMode.Info.Error := autoEXECUTE_PROGRAM_ERROR;
				AutoMode.Info.CurrentState := autoSTATE_ERROR;
				AutoMode.Parameters.Execute := FALSE;
				AutoMode.Parameters.Continuous := FALSE;
			END_IF
			(*RoboArmPara.ProgramName := AutoMode.Parameters.ProgramName;
			RoboArm.Update := TRUE;
			RoboArm.MoveProgram := TRUE;
			IF RoboArm.MoveDone THEN
				RoboArm.MoveProgram := FALSE;
			END_IF*)

		autoSTATE_DONE: //this state is a goto for execute when it's done

			IF NOT AutoMode.Parameters.Continuous THEN //if Continuous isn't set, return to idle
				AutoMode.Parameters.Execute := FALSE;
				AutoMode.Info.CurrentState := autoSTATE_WAIT;
			ELSE //do it as long as Continuous is set or until Abort isn't set
				AutoMode.Parameters.Execute := TRUE;
				AutoMode.Info.CurrentState := autoSTATE_EXECUTE;
			END_IF
				//AutoMode.Info.CurrentState := autoSTATE_WAIT;
			AutoMode.Cmds.UnloadProgram(Execute := FALSE); //just a precaution
			AutoMode.Cmds.LoadProgram(Execute := FALSE);
			AutoMode.Cmds.ExecuteProgram(Execute := FALSE);

		autoSTATE_PAUSE: //this state pauses active program execution
			IF AutoMode.Cmds.PauseProgram.Done THEN
				AutoMode.Cmds.PauseProgram.Execute := FALSE;
				AutoMode.Cmds.PauseProgram();
				AutoMode.Parameters.Pause := FALSE;
				AutoMode.Info.Paused := TRUE;
				AutoMode.Info.CurrentState := autoSTATE_WAIT;
			ELSIF AutoMode.Cmds.PauseProgram.Error THEN
				AutoMode.Info.IsError := TRUE;
				AutoMode.Info.Error := autoPAUSE_ERROR;
				AutoMode.Info.ErrorID := AutoMode.Cmds.PauseProgram.ErrorID;
				AutoMode.Info.CurrentState := autoSTATE_ERROR;
			ELSE

				AutoMode.Cmds.PauseProgram(AxesGroup := ADR(AxesGroup), Execute := TRUE);
			END_IF

		autoSTATE_CONTINUE: //this state continues paused program
			IF AutoMode.Cmds.ContinueProgram.Done THEN
				AutoMode.Cmds.ContinueProgram.Execute := FALSE;
				AutoMode.Cmds.ContinueProgram();
				AutoMode.Parameters.Continue := FALSE;
				AutoMode.Info.Paused := FALSE;
				AutoMode.Info.CurrentState := autoSTATE_WAIT;
			ELSIF AutoMode.Cmds.ContinueProgram.Error THEN
				AutoMode.Info.IsError := TRUE;
				AutoMode.Info.Error := autoCONTINUE_ERROR;
				AutoMode.Info.ErrorID := AutoMode.Cmds.ContinueProgram.ErrorID;
				AutoMode.Info.CurrentState := autoSTATE_ERROR;
			ELSE
				AutoMode.Cmds.ContinueProgram(AxesGroup := ADR(AxesGroup), Execute := TRUE);
			END_IF

		autoSTATE_ABORT: //a noncritical stop
			IF AutoMode.Cmds.GroupStop.Done THEN //it's stopped
				AutoMode.Cmds.GroupStop.Execute := FALSE;
				AutoMode.Cmds.GroupStop();
				AutoMode.Parameters.Execute := FALSE;
				AutoMode.Parameters.Unload := FALSE;
				//AutoMode.Parameters.Load := TRUE; //for some reason loading a program after stopping is good.
				AutoMode.Parameters.Abort := FALSE;
				AutoMode.Parameters.Continuous := FALSE;
				AutoMode.Info.Paused := FALSE;
				AutoMode.Info.CurrentState := autoSTATE_WAIT;

			ELSIF AutoMode.Cmds.GroupStop.Error THEN
				AutoMode.Info.IsError := TRUE;
				AutoMode.Info.Error := autoABORT_ERROR;
				AutoMode.Info.ErrorID := AutoMode.Cmds.GroupStop.ErrorID;
				AutoMode.Info.CurrentState := autoSTATE_ERROR;
			ELSE

				AutoMode.Cmds.GroupStop(AxesGroup := ADR(AxesGroup), Execute := TRUE, StopMode := mcSTOPMODE_JERK_LIMIT); //take into account jerk limit as it's a noncritical stop
			END_IF

			//D edit
			AutoMode.Parameters.Abort:=FALSE;

		autoSTATE_ERROR: //error state, ErrorReset is reset automatically. reset state control variables
			AutoMode.Info.IsError := TRUE;
			AutoMode.Parameters.Execute := FALSE;
			AutoMode.Parameters.Unload := FALSE;
			AutoMode.Parameters.Load := FALSE;
			AutoMode.Parameters.Continuous := FALSE;

			IF AutoMode.Parameters.ErrorReset THEN
				AutoMode.Info.Error := autoNO_ERROR;
				AutoMode.Info.ErrorID := 0;

			END_IF

			IF AutoMode.Info.ErrorID = 0 THEN
				AutoMode.Info.IsError := FALSE;
				AutoMode.Parameters.ErrorReset := FALSE;
				AutoMode.Info.CurrentState := autoSTATE_WAIT;
			END_IF

	END_CASE

END_FUNCTION_BLOCK
```

#### R3BrakeSet.st
```iecst
(* TODO: Add your comment here *)
FUNCTION_BLOCK R3BrakeSet
	(* SEE: 45ae2aa8-d38d-40c1-866a-6c119063ad8e for information on group brake control for Comau Racer 3 robot *)
	//these settings are set to default values, may be changed later if needed.
	BrakePara.AutomaticControl := mcSWITCH_ON;
	BrakePara.AutomaticInductionStop := mcSWITCH_OFF;
	BrakePara.ControlMonitoring := mcSWITCH_OFF; //changed, it's a game changer.
	BrakePara.EnableSBTRequestBySMC := mcSWITCH_OFF;
	BrakePara.MovementMonitoring := mcSWITCH_ON;
	BrakePara.RestrictedBrakeControl := mcSWITCH_OFF; //changed, it's a game changer.
	BrakePara.TestAtPowerOff := mcSWITCH_OFF;
	BrakePara.TestAtPowerOn := mcSWITCH_OFF;
	BrakePara.VoltageMonitoring := mcSWITCH_ON;
	BrakePara.ControlMonitoringFilterTime := 0.5;
	BrakeSet.Parameters := BrakePara;

	IF CurrentAxis = 1 THEN
		BrakeSet.Axis := ADR(Axis1);
		BrakeSet.Execute := TRUE;
		IF BrakeSet.Done THEN
			BrakeSet.Execute := FALSE;
			CurrentAxis := CurrentAxis + 1;
		END_IF
		BrakeSet();
	ELSIF CurrentAxis = 2 THEN
		BrakeSet.Axis := ADR(Axis2);
		BrakeSet.Execute := TRUE;
		IF BrakeSet.Done THEN
			BrakeSet.Execute := FALSE;
			CurrentAxis := CurrentAxis + 1;
		END_IF
		BrakeSet();
	ELSIF CurrentAxis = 3 THEN
		BrakeSet.Axis := ADR(Axis3);
		BrakeSet.Execute := TRUE;
		IF BrakeSet.Done THEN
			BrakeSet.Execute := FALSE;
			CurrentAxis := CurrentAxis + 1;
		END_IF
		BrakeSet();
	ELSIF CurrentAxis = 4 THEN
		BrakeSet.Axis := ADR(Axis4);
		BrakeSet.Execute := TRUE;
		IF BrakeSet.Done THEN
			BrakeSet.Execute := FALSE;
			CurrentAxis := CurrentAxis + 1;
		END_IF
		BrakeSet();
	ELSIF CurrentAxis = 5 THEN
		BrakeSet.Axis := ADR(Axis5);
		BrakeSet.Execute := TRUE;
		IF BrakeSet.Done THEN
			BrakeSet.Execute := FALSE;
			CurrentAxis := CurrentAxis + 1;
		END_IF
		BrakeSet();
	ELSIF CurrentAxis = 6 THEN
		BrakeSet.Axis := ADR(Axis6);
		BrakeSet.Execute := TRUE;
		IF BrakeSet.Done THEN
			BrakeSet.Execute := FALSE;
			CurrentAxis := CurrentAxis + 1;
		END_IF
		BrakeSet();
	ELSIF CurrentAxis = 7 THEN
		Done := TRUE;
	END_IF

END_FUNCTION_BLOCK
```

#### R3Workspace.st
```iecst
(* TODO: Add your comment here *)
FUNCTION_BLOCK R3Workspace
	(*Para.Para.ModalDataBehaviour := mcAGFMDB_USE_AX_GRP_SET
	Para.Para.SelfCollisionDetection := mcAGFWSCD_EN;
	Para.Para.WorkspaceReference.Name := 'R3WorkSpace';*)

	Para.Cmd.Name := 'Feature_WorkspaceMonitoring';
	Para.Cmd.DataType := mcCFG_AXGRP_FEAT_WSM;
	Para.Cmd.DataAddress := ADR(Para.Para);
	Para.Cmd.Execute := TRUE;
	Para.Cmd();

	IF Para.Cmd.Done THEN
		Para.Done := TRUE;
		Para.Cmd.Execute := FALSE;
		Para.Cmd();
	END_IF

END_FUNCTION_BLOCK
```

#### AxisControl.fun - not listed in the package file held
```iecst
(*
steruje zmianami osi zadanymi w ManualControl.AxisControl.axis1-6
 zwraca 1 gdy się wykona
 docelowo będzie używane w głównym stanie "READY"
 *)
FUNCTION AxisControl : BOOL
	VAR_INPUT
		axis1:UDINT;
		axis2:UDINT;
		axis3:UDINT;
		axis4:UDINT;
		axis5:UDINT;
		axis6:UDINT;
	END_VAR

	VAR
		AxisControlState : AxisControlStateType;
	END_VAR
```

#### Action.st - not listed in the package file held
```iecst
ACTION Action:

END_ACTION
```

#### ManualMode.st - not listed in the package file held
```iecst
ACTION ManualMode:

	IF ManualModePara.Direction = POSITIVE THEN // set actual axis velocity based on which direction it's set to be moved
		ManualModePara.JogVelocityActual := ManualModePara.JogVelocity;
	ELSIF ManualModePara.Direction = NEGATIVE THEN
		ManualModePara.JogVelocityActual := -1 * ManualModePara.JogVelocity;
	END_IF

	RoboArmPara.Jog.CoordSystem := ManualModePara.CoordinateSystem;
	RoboArmPara.Jog.PathLimits := ManualModePara.PathLimits;

	IF ManualModePara.AxisButton.Q1 THEN // if a button is pressed, write corresponding velocity to the jog velocity array
		RoboArmPara.Jog.Velocity[0] := ManualModePara.JogVelocityActual;
		RoboArm6Axis.Jog := TRUE;
	ELSIF ManualModePara.AxisButton.Q2 THEN
		RoboArmPara.Jog.Velocity[1] := ManualModePara.JogVelocityActual;
		RoboArm6Axis.Jog := TRUE;
	ELSIF ManualModePara.AxisButton.Q3 THEN
		RoboArmPara.Jog.Velocity[2] := ManualModePara.JogVelocityActual;
		RoboArm6Axis.Jog := TRUE;
	ELSIF ManualModePara.AxisButton.Q4 THEN
		RoboArmPara.Jog.Velocity[3] := ManualModePara.JogVelocityActual;
		RoboArm6Axis.Jog := TRUE;
	ELSIF ManualModePara.AxisButton.Q5 THEN
		RoboArmPara.Jog.Velocity[4] := ManualModePara.JogVelocityActual;
		RoboArm6Axis.Jog := TRUE;
	ELSIF ManualModePara.AxisButton.Q6 THEN
		RoboArmPara.Jog.Velocity[5] := ManualModePara.JogVelocityActual;
		RoboArm6Axis.Jog := TRUE;
	ELSE //if no buttons are pressed reset jog velocity array
		RoboArm6Axis.Jog := FALSE;
		FOR j := 0 TO 5 BY 1 DO //set every jog velocity to 0
			RoboArmPara.Jog.Velocity[j] := 0.0;
		END_FOR;
	END_IF

END_ACTION
```

#### R3Brake.st - not listed in the package file held
```iecst
(* TODO: Add your comment here *)
FUNCTION_BLOCK R3Brake

	Brake.Info.Done := FALSE;

	Brake.Parameters := Parameters;

	IF Brake.Parameters.ReadState THEN
		Brake.Info.BrakeOp := mcBRAKE_GET_STATUS;
		Brake.Cmds.BrakeOperation(Axis := ADR(Axis), Execute := TRUE, Command := Brake.Info.BrakeOp);
		IF Brake.Cmds.BrakeOperation.Done THEN
			Brake.Info.BrakeStatus := Brake.Cmds.BrakeOperation.BrakeStatus;
			Brake.Cmds.BrakeOperation.Execute := FALSE;
			Brake.Cmds.BrakeOperation();
			Brake.Parameters.ReadState := FALSE;
			Brake.Info.Done := TRUE;
		END_IF
	END_IF

	Info := Brake.Info;

END_FUNCTION_BLOCK
```

#### Library Logical/Libraries/RacerLib/ManualCtrl (IEC)

##### ManualCtrl.fun - Exported functions and function blocks
```iecst
(*
steruje zmianami osi zadanymi w ManualControl.AxisControl.axis1-6
 zwraca 1 gdy się wykona
 docelowo będzie używane w głównym stanie "READY"
 *)

FUNCTION test : BOOL
	VAR_INPUT
		in2 : INT;
		in3 : INT;
		in1 : INT;
	END_VAR
END_FUNCTION
```

##### TEST.st
```iecst
(* TODO: Add your comment here *)
FUNCTION test
	IF (in1 + in2 + in3) > 15 THEN
		test := TRUE;
	ELSE
		test := FALSE;
	END_IF;
END_FUNCTION
```

##### Action.st
```iecst
ACTION TestAction:

END_ACTION
```

- Visualisation Logical/mappView (not shown)

### Program Logical/Racer3/Control (IEC)

#### Main.st - Init, cyclic, exit code
```iecst
PROGRAM _INIT

	RoboArm6Axis.Enable := TRUE;

	RoboArm6Axis.Override := 100.0; //it's non-100 only for automatic mode
	RoboArm6AxisPara.ProgramName := 'Point.st';    //File stored on FileDevice, default program (Point.st moves TCP to -200, 300, 800)
	RoboArm6Axis.MpLink := ADR(gAxesGroupRacer3);
	RoboArm6Axis.Parameters := ADR(RoboArm6AxisPara);
	RoboArm6AxisPara.Acceleration := 1000.0;
	RoboArm6AxisPara.Deceleration := 1000.0;
	RoboArm6AxisPara.Velocity := 69.0;

	Communication.ReturnToZero := FALSE;
	ManualControlPara.PathLimits.Acceleration := 1000.0;
	ManualControlPara.PathLimits.Deceleration := 1000.0;
	ManualControlPara.PathLimits.Velocity := 150.0;
	ManualControlPara.PathLimits.Jerk := 0.0;
	ManualControlPara.Direction := -1;

	State := STATE_INIT;
	Communication.Power := FALSE;
	i;
	Brakes;

	//FileMgmt(MpLink := ADR(FileManagement), Enable := TRUE, Configuration := ADR(FileMgmtConfig));

	gRacer3HomeRestorePos; //call home restore position variable to init it in memory
	//MpAlarmXCore_Control(MpLink := ADR(gAlarmXCore), Enable := TRUE);

	AutomaticCurrentLanguage; //variable used for changing script language

	RoboArm6Axis();

END_PROGRAM

PROGRAM _CYCLIC

	IF RoboArm6Axis.Error THEN
		State := STATE_ERROR;
	END_IF
	(*
	IF Communication.Stop THEN
		//stops and goes to standby
		RoboArm6Axis.MoveLinear := FALSE;
		RoboArm6Axis.MoveDirect := FALSE;
		RoboArm6Axis.Jog := FALSE;
		SemiAutoControlPara.Flag := FALSE;
		ManualControlPara.ActivateMove:=FALSE;
		//TODO turn off traces from all moves for sure, not only flags (clean them up)
		State:= STATE_READY;
	END_IF
	*)

	IF Communication.WarmRestart THEN
		Communication.Power := FALSE;
		RoboArm6Axis.Power := FALSE;
		Communication.WarmRestart := FALSE;
		SYSreset(1,1);
	END_IF
	UpdateCheck;

	IF NOT Communication.Power AND NOT (State = STATE_BRAKES) THEN //power commands must have no effect in STATE_BRAKES
		//RoboArm6Axis.Power := FALSE;
		GroupPower(AxesGroup := ADR(gAxesGroupRacer3), Enable := FALSE);
		IF NOT GroupPower.Status THEN
			State := STATE_INIT;
		END_IF

	END_IF

	CASE State OF
		STATE_ERROR:
			Communication.txt_State_out:="Error";
			Communication.txt_State_out_front:= '$$IAT/ControlPage/txt_State_out_front.Error';

			GroupPower(AxesGroup := ADR(gAxesGroupRacer3), Enable := FALSE); //this powers off the axes
			ManualControlPara.ExitManual:=FALSE;
			IF GroupReset.Done THEN
				GroupReset.Execute := FALSE;
				GroupReset();
				Communication.ErrorReset := FALSE;
			ELSIF NOT RoboArm6Axis.Error THEN //if there's no error, go to INIT
				RoboArm6Axis.ErrorReset := FALSE;
				State := STATE_INIT;
			ELSIF Communication.ErrorReset THEN
				GroupReset(AxesGroup := ADR(gAxesGroupRacer3), Execute := TRUE);
				RoboArm6Axis.ErrorReset:=TRUE;
			END_IF

		STATE_INIT:
			Communication.txt_State_out:="Initialization";
			Communication.txt_State_out_front:= '$$IAT/ControlPage/txt_State_out_front.Init';
			ManualControlPara.ExitManual := FALSE;
			(*IF RoboArm6Axis.PowerOn THEN
				Communication.Power := TRUE;
				Communication.BrakesSet := TRUE;
				//State := STATE_POWER_ON;
			ELSE*)

			IF NOT Communication.BrakesSet THEN
				SetBrakes.Axis1 := ADR(gAxisQ1);
				SetBrakes.Axis2 := ADR(gAxisQ2);
				SetBrakes.Axis3 := ADR(gAxisQ3);
				SetBrakes.Axis4 := ADR(gAxisQ4);
				SetBrakes.Axis5 := ADR(gAxisQ5);
				SetBrakes.Axis6 := ADR(gAxisQ6);
				SetBrakes();
				IF SetBrakes.Done THEN
					Communication.BrakesSet := TRUE;
				END_IF
				//RoboArm6Axis.Enable := TRUE;

			ELSE //if brake parameters have been set
				// brake operation functions (only when robot is powered off!)
				IF Communication.BrakeClose THEN
					i := 1;
					Brakes.Info.State := brakeCLOSE;
					State := STATE_BRAKES;

				ELSIF Communication.BrakeOpen THEN
					i := 1;
					Brakes.Info.State := brakeOPEN;
					State := STATE_BRAKES;

				ELSIF Communication.BrakeReadStatus THEN
					i := 1;
					Brakes.Info.State := brakeREAD;
					State := STATE_BRAKES;

				ELSIF Communication.Power AND NOT (State = STATE_BRAKES) THEN //power commands have no effect in STATE_BRAKES
					State := STATE_POWER_ON;
				END_IF
				END_IF

		STATE_POWER_ON:
			Communication.txt_State_out:="Power";
			Communication.txt_State_out_front:= '$$IAT/ControlPage/txt_State_out_front.Power';

			IF NOT RoboArm6Axis.PowerOn AND RoboArm6Axis.Info.ReadyToPowerOn THEN
				GroupPower(AxesGroup := ADR(gAxesGroupRacer3), Enable := TRUE);
				//RoboArm6Axis.Power := TRUE;
			END_IF

			IF (GroupPower.Status AND GroupPower.Enable) OR RoboArm6Axis.PowerOn THEN //Status tells whether the group is really powered on, Enable must be true., second condition applies when a transfer is initiated - no real benefit otherwise
				State := STATE_HOMING;
			END_IF

			(*IF RoboArm6Axis.PowerOn THEN //unused
				State := STATE_HOMING;

			END_IF*)

		STATE_HOMING:
			Communication.txt_State_out:="Homing";
			Communication.txt_State_out_front:= '$$IAT/ControlPage/txt_State_out_front.Homing';

			IF gIsCalibrated THEN
				CalibrationStateBtn := FALSE;
				IF RoboArm6Axis.IsHomed THEN //autohoming after power on
					RoboArm6Axis.Home := FALSE;
					State := STATE_READY;
				ELSE

					RoboArm6Axis.Home := TRUE;
					//Calibration.Cmds.GroupHome(AxesGroup := ADR(gAxesGroupRacer3), Execute := TRUE, HomingMode := Calibration.Para.HomingModeEnum);
					(*IF Calibration.Cmds.GroupHome.Done THEN
					State := STATE_READY;
					END_IF*)

				END_IF
			ELSE
				CalibrationStateBtn := TRUE;
				State := STATE_CALIBRATION; //if the system wasn't calibrated before, make it be calibrated
				Calibration.Info.CurrentState := STATE_BEGIN;

			END_IF

		STATE_READY:
			//changeStatePending so change mode is impossible while in-move (before state comes to ready) for example for auto and semiauto
			(*
			IF ControlSelector = ManualJog AND Communication.changeModePending <> 1 THEN
				// exit from MANUAL
				// when exiting ManualMode from mappView bind ManualModePara.ExitMode := TRUE and pending state, both at once
				// because we want to wait till semiAuto and Auto finishes and then goes to READY state, but for manual we have to go out manually
				ManualControlPara.ExitManual := TRUE;
			END_IF
			*)
			(*IF Communication.ReadWorkspace OR R3WorkspaceFB.Para.Cmd.Busy THEN
				WorkspaceControl.Cmd.Mode := mcPCM_LOAD;
				R3WorkspaceFB(Para := WorkspaceControl);
				IF R3WorkspaceFB.Para.Done THEN
					Communication.ReadWorkspace := FALSE;
				END_IF

			END_IF*)

			Communication.ReturnToZero := FALSE; //reset ReturnToZero flag each time manual mode is exit
			(* TODO: Better handling of fake home, do it per axis after each save - DONE*)
			IF NOT Communication.ResetHome THEN //if ResetHome is set off
				IF ControlSelector = ManualJog THEN
					MpAuditWStringChange(MpLink:= gAuditTrailLink, Old := Communication.txt_State_out ,New:="ManualControl", Identifier := 'ControlMode');

					State := STATE_MANUAL_CONTROL;
				ELSIF ControlSelector = SemiAutomatic THEN
					MpAuditWStringChange(MpLink:= gAuditTrailLink, Old :=Communication.txt_State_out,New:="SemiAutoControl", Identifier := 'ControlMode');
					State := STATE_SEMI_AUTOMATIC;
				ELSIF ControlSelector = Automatic THEN
					MpAuditWStringChange(MpLink:= gAuditTrailLink, Old :=Communication.txt_State_out,New:="AutoControl", Identifier := 'ControlMode');
					State := STATE_AUTOMATIC;
				ELSE
					Communication.txt_State_out:="Ready";
					Communication.txt_State_out_front:= '$$IAT/ControlPage/txt_State_out_front.Ready';
				END_IF
			ELSE
				State := STATE_CALIBRATION;
			END_IF

			ControlSelector := Communication.changeModePending;
			// TODO think what happens when ControlSelector changes in-between init,update,start,go in auto and semiauto and fix it
			// maybe do something similar to exit mode in manual

		STATE_MANUAL_CONTROL:
			//Communication.LastControlState := 'Manual';
			//ChangeMode
			ManualControlPara.ExitManual:=FALSE;
			IF ControlSelector = ManualJog AND Communication.changeModePending <> 1 THEN
				// exit from MANUAL
				ManualControlPara.ExitManual :=TRUE;
				ControlSelector := Communication.changeModePending;
				State := STATE_READY;
				//Communication.Stop:=FALSE;
			END_IF
			IF Communication.Stop THEN
				ManualControlPara.ExitManual := TRUE;
				Communication.Stop := FALSE;
			END_IF

			Communication.txt_State_out := "ManualControl";
			Communication.txt_State_out_front := '$$IAT/ControlPage/txt_State_out_front.Manual';
			RoboArm6Axis.Override := 100.0; //required for Jog
			//ManualControlPara.PathLimits.Acceleration;
			//ManualControlPara.PathLimits.Deceleration;
			//ManualControlPara.PathLimits.Jerk;
			ManualControlPara.PathLimits.Velocity := 1000.0;
			//ManualControlPara; //main struct to be bound in mapp view
			IF Communication.ReturnToZero AND ManualControlPara.JogVelocity >= 1.0 THEN //return to Zero function, only works when velocity is greater than 1.0 (otherwise move could not be executed)
				RoboArm6AxisPara.Position := gRacer3ZeroPosition; //read from PV set during calibration
				RoboArm6AxisPara.CoordSystem := 0;
				RoboArm6AxisPara.ManualMoveType := mcMOVE_ABSOLUTE;
				RoboArm6AxisPara.Velocity := ManualControlPara.JogVelocity;
				RoboArm6Axis.MoveDirect := TRUE;
				IF RoboArm6Axis.MoveDone THEN
					RoboArm6Axis.MoveDirect := FALSE;
					Communication.ReturnToZero := FALSE;
				END_IF

			ELSE
				Communication.ReturnToZero := FALSE;
				RoboArm6Axis.MoveDirect := FALSE;
				ManualControl(ManualModePara := ManualControlPara, RoboArm := RoboArm6Axis, RoboArmPara := RoboArm6AxisPara,MainState := State, ControlSelector := ControlSelector);
			END_IF

		STATE_SEMI_AUTOMATIC:
			//Communication.LastControlState := 'SemiAuto';

			//ChangeMode
			IF ControlSelector = SemiAutomatic AND Communication.changeModePending <> 2 THEN
				// exit from SemiAuto
				SemiAutoControlPara.ExitSemiAuto:=TRUE;
				ControlSelector:=Communication.changeModePending;
				State:=STATE_READY;
				//Communication.Stop:=FALSE;
			END_IF
			IF Communication.Stop THEN
				SemiAutoControlPara.ExitSemiAuto:=TRUE;
				Communication.Stop:=FALSE;
			END_IF

			Communication.txt_State_out:="SemiAutoControl";
			Communication.txt_State_out_front:= '$$IAT/ControlPage/txt_State_out_front.SemiAuto';
			RoboArm6Axis.Override := 100.0;
			SemiAutoControl(SemiAutoModePara := SemiAutoControlPara, RoboArm := RoboArm6Axis, RoboArmPara := RoboArm6AxisPara, MainState := State, ControlSelector := ControlSelector);

		STATE_AUTOMATIC:
			//Communication.LastControlState := 'Automatic';
			Communication.txt_State_out:="AutoControl";
			Communication.txt_State_out_front:= '$$IAT/ControlPage/txt_State_out_front.Auto';

			IF ControlSelector = Automatic AND Communication.changeModePending <> 3 THEN
				// exit from Auto
				AutomaticModePara.Parameters.Abort:=TRUE;
				ControlSelector:=Communication.changeModePending;
				State:=STATE_READY;
			END_IF
			(*IF Communication.Pause AND NOT Communication.Stop THEN
				AutomaticModePara.Parameters.Pause:=TRUE;
			END_IF
			IF NOT Communication.Pause AND AutomaticModePara.Parameters.Pause AND NOT Communication.Stop THEN
				AutomaticModePara.Parameters.Continue:=TRUE;
			END_IF
			IF Communication.Stop THEN
				AutomaticModePara.Parameters.Abort:=TRUE;
				Communication.Stop:=FALSE;
			END_IF

			AutomaticModePara.Parameters;
			AutomaticModePara.Parameters.ProgramName;
			//AutomaticModePara.Parameters.Execute := TRUE;
			//AutomaticModePara.Info.CurrentState := autoSTATE_WAIT;
			AutomaticMode(AutoMode := AutomaticModePara, AxesGroup := ADR(gAxesGroupRacer3));*)
			PathName;
			FileName;
			IF AutomaticCurrentLanguage THEN

				AutomaticModePara.Parameters;
				AutomaticModePara.Parameters.ProgramName := FileName;
				//AutomaticModePara.Parameters.Execute := TRUE;
				//AutomaticModePara.Info.CurrentState := autoSTATE_WAIT;
				AutomaticMode(AutoMode := AutomaticModePara, AxesGroup := ADR(gAxesGroupRacer3));

				//AutomaticModePara.Cmds.ExecuteProgram(AxesGroup := ADR(gAxesGroupRacer3), Execute := TRUE, Name := AutomaticModePara.Parameters.ProgramName);
			ELSE
				//everything here happens in the widget
			END_IF

		STATE_CALIBRATION:

			//perform initial homing to trick ACOPOS into thinking axes are homed, basically set home to current position.
			CalibrationAction;

			Communication.txt_State_out:="Calibration";
			Communication.txt_State_out_front:= '$$IAT/ControlPage/txt_State_out_front.Calibration';

		STATE_BRAKES:
			//Brakes.Cmds.BrakeOperation.SelectMode := 0;
			IF Brakes.Cmds.BrakeOperation.Error THEN
				Brakes.Info.State := brakeERROR;
			ELSE
				Brakes.Info.Error := FALSE;
			END_IF

			CASE Brakes.Info.State OF
				brakeERROR:
					Communication.BrakeClose := FALSE;
					Communication.BrakeOpen := FALSE;
					Communication.BrakeReadStatus := FALSE;
					Brakes.Cmds.BrakeOperation.Execute := FALSE;
					Brakes.Info.Error := TRUE;
					Brakes.Cmds.BrakeOperation();
					State := STATE_INIT;
				brakeDONE:
					Brakes.Cmds.BrakeOperation.Execute := FALSE;

					Brakes.Cmds.BrakeOperation();
					State := STATE_INIT;

				brakeOPEN:
					Communication.BrakeOpen := FALSE;
					Brakes.Cmds.BrakeOperation.AxesGroup := ADR(gAxesGroupRacer3);
					Brakes.Parameters.BrakeCmd := mcBRAKE_OPEN;
					IF Brakes.Cmds.BrakeOperation.Done AND (i = 1) THEN
						Brakes.Cmds.BrakeOperation.Execute := FALSE;
						Brakes.Cmds.BrakeOperation();
						i := 2;
					ELSIF Brakes.Cmds.BrakeOperation.Done AND (i = 2) THEN
						Brakes.Cmds.BrakeOperation.Execute := FALSE;
						Brakes.Cmds.BrakeOperation();
						i := 3;
						Communication.BrakeReadStatus := TRUE;
						Brakes.Info.State := brakeDONE;
					ELSIF (i < 3) THEN
						Brakes.Cmds.BrakeOperation.Command := Brakes.Parameters.BrakeCmd;
						Brakes.Cmds.BrakeOperation.Identifier := i;
						Brakes.Cmds.BrakeOperation.Execute := TRUE;

						Brakes.Cmds.BrakeOperation();
					END_IF

				brakeCLOSE:
					Communication.BrakeClose := FALSE;
					Brakes.Cmds.BrakeOperation.AxesGroup := ADR(gAxesGroupRacer3);
					Brakes.Parameters.BrakeCmd := mcBRAKE_CLOSE;
					IF Brakes.Cmds.BrakeOperation.Done AND (i = 1) THEN
						Brakes.Cmds.BrakeOperation.Execute := FALSE;
						Brakes.Cmds.BrakeOperation();
						i := 2;
					ELSIF Brakes.Cmds.BrakeOperation.Done AND (i = 2) THEN
						Brakes.Cmds.BrakeOperation.Execute := FALSE;
						Brakes.Cmds.BrakeOperation();
						i := 3;
						Communication.BrakeReadStatus := TRUE;
						Brakes.Info.State := brakeDONE;
					ELSIF (i < 3) THEN
						Brakes.Cmds.BrakeOperation.Command := Brakes.Parameters.BrakeCmd;
						Brakes.Cmds.BrakeOperation.Identifier := i;
						Brakes.Cmds.BrakeOperation.Execute := TRUE;

						Brakes.Cmds.BrakeOperation();
					END_IF

				brakeREAD:
					Communication.BrakeReadStatus := FALSE;
					Brakes.Parameters.BrakeCmd := mcBRAKE_GET_STATUS;
					Brakes.Cmds.BrakeOperation.AxesGroup := ADR(gAxesGroupRacer3);
					IF Brakes.Cmds.BrakeOperation.Done AND (i = 1) THEN
						Brakes.Info.BrakeStatus[i] := Brakes.Cmds.BrakeOperation.BrakeStatus;
						Brakes.Cmds.BrakeOperation.Execute := FALSE;
						Brakes.Cmds.BrakeOperation();
						i := 2;
					ELSIF Brakes.Cmds.BrakeOperation.Done AND (i = 2) THEN
						Brakes.Info.BrakeStatus[i] := Brakes.Cmds.BrakeOperation.BrakeStatus;
						Brakes.Cmds.BrakeOperation.Execute := FALSE;
						Brakes.Cmds.BrakeOperation();
						i := 3;
						Brakes.Info.State := brakeDONE;
					ELSIF (i < 3) THEN
						Brakes.Cmds.BrakeOperation.Command := Brakes.Parameters.BrakeCmd;
						Brakes.Cmds.BrakeOperation.Identifier := i;
						Brakes.Cmds.BrakeOperation.Execute := TRUE;

						Brakes.Cmds.BrakeOperation();
					END_IF

				END_CASE

	END_CASE

	RoboArm6Axis();

	////////////Visualization Variables/////////////
	VisAction;

END_PROGRAM

PROGRAM _EXIT
	(* Insert code here *)
	RoboArm6Axis.Power := FALSE;
	RoboArm6Axis.Enable := FALSE;

	RoboArm6Axis(); //this will free up MpLink (possibly)
END_PROGRAM
```

#### Types.typ - Local data types
```iecst
(*
TYPE
	ControlSelectEnum :
		(
		ManualJog,
		SemiAutomatic,
		Automatic
		);
	CalibrationType : 	STRUCT
		Info : CalibrationInfo; (*Information portion of calibration.*)
		Cmds : CalibrationCmds; (*Calibration commands*)
		Para : CalibrationPara; (*Calibration parameters*)
	END_STRUCT;
	CalibrationPara : 	STRUCT
		Parameters : R3CalibrationType;
		HomingParameters : McAcpAxHomingParType;
		FakeHomingModeEnum : ARRAY[0..14]OF McHomingModeEnum := [15(mcHOMING_DIRECT)];
		Positions : ARRAY[0..14]OF LREAL := [15(0.0)];
		HomingModeEnum : ARRAY[0..14]OF McHomingModeEnum := [15(mcHOMING_INIT)];
	END_STRUCT;
	CalibrationCmds : 	STRUCT
		Mode : R3CalibrationMode;
		InitHome : MC_BR_InitHome_AcpAx;
		GroupHome : MC_BR_GroupHome_15;
	END_STRUCT;
	CalibrationInfo : 	STRUCT
		CurrentState : OuterCalibrationState;
	END_STRUCT;
	OuterCalibrationState :
		(
		STATE_BEGIN,
		STATE_FAKE_HOME,
		STATE_MOVING,
		STATE_SAVING_POSITION,
		STATE_DONE
		);
END_TYPE
*)
```

#### Variables.var - Local variables
```iecst
VAR
	BrakeStatus : ARRAY[0..5] OF McBrakeStatusEnum; (*Brake information*)
	Brakes : R3BrakeType;
	KeyCheck : R3KeyCheckType;
	AutomaticCurrentLanguage : BOOL; (*selects which language to use (0 - G-Code, 1 - ST)*)
	AutomaticMode : R3AutomaticMode; (*automatic mode FB*)
	AutomaticModePara : R3AutomaticModeType; (*Main automatic mode variable*)
	RoboArm6AxisPara : MpRoboArm6AxisParType; (*This variable defines parameters of the robot*)
	RoboArm6Axis : MpRoboArm6Axis; (*This is the robot in question*)
	State : R3StateMachineEnum;
	ControlSelector : ControlSelectEnum := None;
	ManualControl : R3ManualMode;
	ManualControlPara : R3ManualModeType;
	i : USINT; (*Counter.*)
	Axis5Calibrated : BOOL; (*If value TRUE then axis 6 can be calibrated*)
	Axis_1to4_calibrated : BOOL; (*If value TRUE then axis 5 can be calibrated*)
	Calibration : R3CalibrationMainType; (*Main calibration variable.*)
	WorkspaceControl : R3WorkspaceType;
	SemiAutoControl : R3SemiAutoMode;
	SemiAutoControlPara : R3SemiAutoModeType;
	MpAlarmXCore_Control : MpAlarmXCore;
	LastState : R3StateMachineEnum; (*Stores last machine state.*)
	CalibrationStateBtn : BOOL; (*TRUE when in state STATE_CALIBRATION *)
	Communication : CommunicationType;
	PathName : STRING[260];
	FileName : STRING[260];
	GroupPower : MC_BR_GroupPower;
	GroupReset : MC_GroupReset;
	SetBrakes : R3BrakeSet; (*Setting brake parameters*)
	R3WorkspaceFB : R3Workspace;
END_VAR
```

#### UpdateCheck.st
```iecst
ACTION UpdateCheck:
	IF Communication.CoordinateSystemSemiAuto THEN //Coordinate system in ManualControl and SemiAutoControl: 9-global  0-axis
		//ManualControlPara.CoordinateSystem := 9;
		IF SemiAutoControlPara.CoordinateSystem <> 9 THEN
			SemiAutoControlPara.CoordinateSystem := 9;
			SemiAutoControlPara.UpdatePending := TRUE;
		END_IF
	ELSE
		//ManualControlPara.CoordinateSystem := 0;
		IF SemiAutoControlPara.CoordinateSystem <> 0 THEN
			SemiAutoControlPara.CoordinateSystem := 0;
			SemiAutoControlPara.UpdatePending := TRUE;
		END_IF
	END_IF

	IF Communication.CoordinateSystemManual THEN //Coordinate system in ManualControl and SemiAutoControl: 9-global  0-axis
		ManualControlPara.CoordinateSystem := 9;
	ELSE
		ManualControlPara.CoordinateSystem := 0;
	END_IF

	IF SemiAutoControlPara.PathMode <> Communication.PathSystem THEN
		SemiAutoControlPara.PathMode := Communication.PathSystem;
		SemiAutoControlPara.UpdatePending :=TRUE;
		// TODO Auto too
	END_IF

	IF SemiAutoControlPara.Mode <> Communication.ModeSystem THEN
		SemiAutoControlPara.Mode := Communication.ModeSystem;
		SemiAutoControlPara.UpdatePending :=TRUE;
		// TODO Auto too
	END_IF
	(*
	IF RoboArm6AxisPara.Distance[0] <>  SemiAutoControlPara.AskedValue.Q0 OR RoboArm6AxisPara.Distance[1] <>  SemiAutoControlPara.AskedValue.Q1 OR RoboArm6AxisPara.Distance[2] <>  SemiAutoControlPara.AskedValue.Q2 OR RoboArm6AxisPara.Distance[3] <>  SemiAutoControlPara.AskedValue.Q3 OR RoboArm6AxisPara.Distance[4] <>  SemiAutoControlPara.AskedValue.Q4 OR RoboArm6AxisPara.Distance[5] <>  SemiAutoControlPara.AskedValue.Q5  OR RoboArm6AxisPara.Position[0] <>  SemiAutoControlPara.AskedValue.Q0 OR RoboArm6AxisPara.Position[1] <>  SemiAutoControlPara.AskedValue.Q1 OR RoboArm6AxisPara.Position[2] <>  SemiAutoControlPara.AskedValue.Q2 OR RoboArm6AxisPara.Position[3] <>  SemiAutoControlPara.AskedValue.Q3 OR RoboArm6AxisPara.Position[4] <>  SemiAutoControlPara.AskedValue.Q4 OR RoboArm6AxisPara.Position[5] <>  SemiAutoControlPara.AskedValue.Q5 THEN
		SemiAutoControlPara.UpdatePending :=TRUE;

	END_IF
	*)
	IF Communication.UpdateSemiAutoVars THEN
		SemiAutoControlPara.UpdatePending :=TRUE;
		Communication.UpdateSemiAutoVars := FALSE;
	END_IF

END_ACTION
```

#### Calibration.st
```iecst
ACTION CalibrationAction:
	IF Communication.ResetHome THEN //this enables the user to reset each axis to 0.0 in software - allows for movement when a (false) workspace violation is set off during calibration.
		Calibration.Info.CurrentState := STATE_FAKE_HOME;
	END_IF

	IF Calibration.Cmds.GroupHome.Done OR NOT Calibration.Cmds.GroupHome.Busy THEN
		Calibration.Cmds.GroupHome.Execute := FALSE;
		Calibration.Cmds.GroupHome();
	END_IF

	CASE Calibration.Info.CurrentState OF
		STATE_BEGIN:
			IF gIsCalibrated THEN
				Calibration.Info.CurrentState := STATE_DONE;
			ELSE

			Calibration.Para.Parameters.CalibrationModePara.JogVelocity := 5.0; //default velocity
			IF RoboArm6Axis.IsHomed AND NOT Communication.ResetHome THEN
				Calibration.Info.CurrentState := STATE_MOVING; //if a home is set, go directly to manual calibration (perhaps calibration on demand?)
			ELSE
				Calibration.Info.CurrentState := STATE_FAKE_HOME; //otherwise set a fake home
				END_IF
			END_IF

		STATE_FAKE_HOME:

			FOR i := 0 TO 5 BY 1 DO
				IF i = 2 THEN
					Calibration.Para.Positions[i] := -90.0; //axis 3 default position is -90.0 degrees
				ELSE
					Calibration.Para.Positions[i] := 0.0;
				END_IF

			END_FOR

			Calibration.Cmds.GroupHome(AxesGroup := ADR(gAxesGroupRacer3), Execute := TRUE, Position := Calibration.Para.Positions, HomingMode := Calibration.Para.FakeHomingModeEnum); //this makes the robot think its axes are 0.0
			IF Calibration.Cmds.GroupHome.Done THEN
				Calibration.Cmds.GroupHome.Execute := FALSE;
				Calibration.Cmds.GroupHome();
				IF Communication.ResetHome THEN //if manual homing reset
					Calibration.Info.CurrentState := STATE_BEGIN;
					Communication.ResetHome := FALSE;
				ELSE
					Calibration.Info.CurrentState := STATE_MOVING;
				END_IF

			END_IF

		STATE_MOVING:

			Calibration.Para.Parameters.CalibrationModePara.PathLimits.Acceleration := 1000.0; //set low acceleration, deceleration and velocity limits for calibration purposes
			Calibration.Para.Parameters.CalibrationModePara.PathLimits.Deceleration := 1000.0;
			//CalibrationModePara.CalibrationModePara.PathLimits.Jerk := 1000.0; //no need to limit jerk
			Calibration.Para.Parameters.CalibrationModePara.PathLimits.Velocity := 100.0;
			//Calibration.Para.Parameters.Axis5to6Para.Axis5Angle := -118.0; //angle defined in calibration pdf (see page 100 of _lb-rc-RACER3-STM_en)
			Calibration.Para.Parameters.Axis5To6Para.AxisMoveVelocity := Calibration.Para.Parameters.CalibrationModePara.JogVelocity; //use low velocity for moving axis 5 for calibrating axis 6
			Calibration.Para.Parameters.CalibrationModePara.CoordinateSystem := 0; //set axis coordinate system for calibration
			//CalibrationModePara.CalibrationState := STATE_START; //reset calibration state everytime after jog

			//Block below send axis references to FB (for inithome)
			Calibration.Para.Parameters.AxesRef[0] := ADR(gAxisQ1);
			Calibration.Para.Parameters.AxesRef[1] := ADR(gAxisQ2);
			Calibration.Para.Parameters.AxesRef[2] := ADR(gAxisQ3);
			Calibration.Para.Parameters.AxesRef[3] := ADR(gAxisQ4);
			Calibration.Para.Parameters.AxesRef[4] := ADR(gAxisQ5);
			Calibration.Para.Parameters.AxesRef[5] := ADR(gAxisQ6);

			Calibration.Cmds.Mode(CalibrationPara := Calibration.Para.Parameters, RoboArm := RoboArm6Axis, RoboArmPara := RoboArm6AxisPara); //call FB with set values

			IF Calibration.Para.Parameters.Axis5To6Para.Axis35Restored AND Calibration.Para.Parameters.AxisCalibrated[5] THEN
				Calibration.Info.CurrentState := STATE_SAVING_POSITION;
				Calibration.Para.Parameters.Axis5To6Para.Axis35Restored := FALSE;
				i := 1;
			END_IF

		STATE_SAVING_POSITION:

			gRacer3ZeroPosition := Calibration.Para.Parameters.SavedPositions; //saving calibrated joint values to PV, might be used for zeroing robot position.

			//common values used for homing, will be saved under gRacer3HomeRestorePos[0..5]
			Calibration.Para.HomingParameters.HomingMode := mcHOMING_RESTORE_POSITION;
			Calibration.Para.HomingParameters.RestorePositionVariableAddress; //SET FOR EVERY AXIS SEPARATELY!

			//save positions to PV
			IF i = 1 THEN
				Calibration.Para.HomingParameters.RestorePositionVariableAddress := ADR(gRacer3HomeRestorePos[0]);
				Calibration.Cmds.InitHome(Axis := ADR(gAxisQ1), Execute := TRUE, HomingParameters := Calibration.Para.HomingParameters);
				IF Calibration.Cmds.InitHome.Done THEN
					i := 2;
				END_IF

			ELSIF i = 2 THEN
				Calibration.Para.HomingParameters.RestorePositionVariableAddress := ADR(gRacer3HomeRestorePos[1]);
				Calibration.Cmds.InitHome(Axis := ADR(gAxisQ2), Execute := TRUE, HomingParameters := Calibration.Para.HomingParameters);
				IF Calibration.Cmds.InitHome.Done THEN
					i := 3;
				END_IF

			ELSIF i = 3 THEN
				Calibration.Para.HomingParameters.RestorePositionVariableAddress := ADR(gRacer3HomeRestorePos[2]);
				Calibration.Cmds.InitHome(Axis := ADR(gAxisQ3), Execute := TRUE, HomingParameters := Calibration.Para.HomingParameters);
				IF Calibration.Cmds.InitHome.Done THEN
					i := 4;
				END_IF

			ELSIF i = 4 THEN
				Calibration.Para.HomingParameters.RestorePositionVariableAddress := ADR(gRacer3HomeRestorePos[3]);
				Calibration.Cmds.InitHome(Axis := ADR(gAxisQ4), Execute := TRUE, HomingParameters := Calibration.Para.HomingParameters);
				IF Calibration.Cmds.InitHome.Done THEN
					i := 5;
				END_IF

			ELSIF i = 5 THEN
				Calibration.Para.HomingParameters.RestorePositionVariableAddress := ADR(gRacer3HomeRestorePos[4]);
				Calibration.Cmds.InitHome(Axis := ADR(gAxisQ5), Execute := TRUE, HomingParameters := Calibration.Para.HomingParameters);
				IF Calibration.Cmds.InitHome.Done THEN
					i := 6;
				END_IF

			ELSIF i = 6 THEN
				Calibration.Para.HomingParameters.RestorePositionVariableAddress := ADR(gRacer3HomeRestorePos[5]);
				Calibration.Cmds.InitHome(Axis := ADR(gAxisQ6), Execute := TRUE, HomingParameters := Calibration.Para.HomingParameters);
				IF Calibration.Cmds.InitHome.Done THEN
					gIsCalibrated := TRUE;
					Calibration.Info.CurrentState := STATE_DONE;
				END_IF

			END_IF

		STATE_DONE:
			//gRacer3BasePosition := RoboArm6Axis.Info.JointAxisPosition; //replaced by assignment at the beginning of STATE_SAVING_POSITIONS

			State:=STATE_HOMING;

	END_CASE
END_ACTION
```

#### VisAction.st
```iecst
ACTION VisAction:
	Communication.NOTCoordinateSystemSemiAuto := NOT Communication.CoordinateSystemSemiAuto;
	Communication.NOTPathSystem	:= NOT Communication.PathSystem;
	Communication.NOTModeSystem := NOT Communication.ModeSystem;

	IF Calibration.Para.Parameters.AxisCalibrated[0] AND Calibration.Para.Parameters.AxisCalibrated[1] AND Calibration.Para.Parameters.AxisCalibrated[2] AND Calibration.Para.Parameters.AxisCalibrated[3] THEN
		Axis_1to4_calibrated := TRUE;
	ELSE
		Axis_1to4_calibrated := FALSE;
	END_IF

	IF Axis_1to4_calibrated AND Calibration.Para.Parameters.AxisCalibrated[4] THEN
		Axis5Calibrated := TRUE;
	ELSE
		Axis5Calibrated := FALSE;
	END_IF

	IF KeyCheck.value_changed AND KeyCheck.event_achieved THEN
		KeyCheck.value_changed := FALSE;
		KeyCheck.event_achieved := FALSE;
	ELSIF KeyCheck.value_changed THEN
		IF KeyCheck.temp_value = KeyCheck.original_combo[KeyCheck.i] THEN
			KeyCheck.pending_combo[KeyCheck.i] := KeyCheck.temp_value;
			KeyCheck.i := KeyCheck.i + 1;
			KeyCheck.value_changed := FALSE;
			IF KeyCheck.i = 6 THEN
				//meets its end
				//make event happen
				KeyCheck.event_achieved := TRUE;
			END_IF
		ELSIF KeyCheck.temp_value <> KeyCheck.pending_combo[KeyCheck.i] THEN
			KeyCheck.i:=0;
		END_IF
	END_IF

	IF Calibration.Para.Parameters.CalibrationModePara.AxisButton.Q1 THEN
		Communication.CalibrationImage := 'Media/calibration/calib_axis1.PNG';
		Communication.TextManager.CalibHelper := '$$IAT/ControlPage/Calibration.Helper.1';
	ELSIF Calibration.Para.Parameters.CalibrationModePara.AxisButton.Q2 THEN
		Communication.CalibrationImage := 'Media/calibration/calib_axis2.PNG';
		Communication.TextManager.CalibHelper := '$$IAT/ControlPage/Calibration.Helper.2';
	ELSIF Calibration.Para.Parameters.CalibrationModePara.AxisButton.Q3 THEN
		Communication.CalibrationImage := 'Media/calibration/calib_axis3.PNG';
		Communication.TextManager.CalibHelper := '$$IAT/ControlPage/Calibration.Helper.3';
	ELSIF Calibration.Para.Parameters.CalibrationModePara.AxisButton.Q4 THEN
		Communication.CalibrationImage := 'Media/calibration/calib_axis4.PNG';
		Communication.TextManager.CalibHelper := '$$IAT/ControlPage/Calibration.Helper.4';
	ELSIF Calibration.Para.Parameters.CalibrationModePara.AxisButton.Q5 THEN
		Communication.CalibrationImage := 'Media/calibration/calib_axis5.PNG';
		Communication.TextManager.CalibHelper := '$$IAT/ControlPage/Calibration.Helper.5';
	ELSIF Calibration.Para.Parameters.CalibrationModePara.AxisButton.Q6 THEN
		Communication.CalibrationImage := 'Media/calibration/calib_axis6.PNG';
		Communication.TextManager.CalibHelper := '$$IAT/ControlPage/Calibration.Helper.6';
	ELSE
		Communication.CalibrationImage := '';
		Communication.TextManager.CalibHelper := '';
	END_IF

	IF Calibration.Para.Parameters.AxisCalibrated[0] AND Calibration.Para.Parameters.AxisCalibrated[1] AND Calibration.Para.Parameters.AxisCalibrated[2] AND Calibration.Para.Parameters.AxisCalibrated[3] AND Calibration.Para.Parameters.AxisCalibrated[4] AND Calibration.Para.Parameters.AxisCalibrated[5] AND NOT gIsCalibrated THEN
		Communication.TextManager.CalibHelper := '$$IAT/ControlPage/Calibration.Helper.7';
		Communication.RestoreAxis5 := TRUE;
	ELSIF gIsCalibrated THEN
		Communication.TextManager.CalibHelper := '$$IAT/ControlPage/Calibration.Helper.8';
		Communication.RestoreAxis5 := FALSE;
	ELSE
		Communication.RestoreAxis5 := FALSE;
	END_IF

	IF Communication.CalibrateAgain THEN

		gIsCalibrated:=FALSE;
		Calibration.Para.Parameters.AxisCalibrated[0] := FALSE;
		Calibration.Para.Parameters.AxisCalibrated[1] := FALSE;
		Calibration.Para.Parameters.AxisCalibrated[2] := FALSE;
		Calibration.Para.Parameters.AxisCalibrated[3] := FALSE;
		Calibration.Para.Parameters.AxisCalibrated[4] := FALSE;
		Calibration.Para.Parameters.AxisCalibrated[5] := FALSE;
		Communication.CalibrateAgain := FALSE;
	END_IF

END_ACTION
```

#### ManualAxisJog.st
```iecst
ACTION ManualAxisMove:

END_ACTION
```

#### Action.st - not listed in the package file held
```iecst
ACTION act1:
c:=a+b;
END_ACTION
```

- Project.language (not shown)

### Program Logical/Auditing (IEC)

#### Variables.var
```iecst
VAR
	TriggerEvent : BOOL;
	TypeVar : WSTRING[100] := "Type";
	MessageVar : WSTRING[100] := "Message";
	CommentVar : WSTRING[100] := "Comment";
	CustomEventStatus : DINT;
	MpAuditTrail_0 : MpAuditTrail;
	NewValue : LREAL;
	OldValue : LREAL;
	ClearBufferBool : BOOL;
	PvTest : BOOL;
	Language : STRING[20] := 'pl|metric';
END_VAR
```

#### Main.st
```iecst
PROGRAM _INIT
	MpAuditTrail_0.Enable := TRUE;
	MpAuditTrail_0.MpLink := ADR(gAuditTrailLink);
	MpAuditTrail_0.DeviceName := ADR('AUDIT');
	//MpAuditTrail_0.Language := ADR(Language);
	MpAuditTrail_0();
END_PROGRAM

PROGRAM _CYCLIC

	//MpAuditTrail_0.Enable := TRUE;
	//Triggering User custom event used for testing audit system.
	IF(TriggerEvent)THEN
		CustomEventStatus := MpAuditCustomEvent(MpLink := gAuditTrailLink, Type := TypeVar, Message := MessageVar, Comment := CommentVar);
		//MpAuditStringChange(MpLink:= gAuditTrailLink, Old :='MANUAL',New:='AUTO', Identifier := 'MODE');

		TriggerEvent := FALSE;
	END_IF
	//Cleaning Buffer using ClearBufferBool/ Click button event sets ClearBufferBool value to TRUE.
	IF(ClearBufferBool)THEN
		MpAuditClearBuffer(MpLink := gAuditTrailLink);
		ClearBufferBool := FALSE;
	END_IF

	MpAuditTrail_0();

END_PROGRAM

PROGRAM _EXIT
	MpAuditTrail_0.Enable := FALSE;
	MpAuditTrail_0();
END_PROGRAM
```

### Program Logical/Alarm (IEC)

#### Variables.var
```iecst
VAR
	TriggerAlarm : BOOL;
	MpAlarmXCoreObject : MpAlarmXCore;
	MpAlarmXHistory_0 : MpAlarmXHistory;
	MC_GroupReadError_0 : MC_GroupReadError;
	ErrorID : DINT;
	RecordID : UDINT;
END_VAR
```

#### Main.st
```iecst
PROGRAM _INIT

	MpAlarmXCoreObject(MpLink := ADR(gAlarmXCoreLink) , Enable := FALSE);
	MpAlarmXHistory_0(MpLink := ADR(gAlarmXHistoryLink), DeviceName := ADR('AUDIT'), Enable := FALSE);

END_PROGRAM

PROGRAM _CYCLIC

	MpAlarmXCoreObject(Enable := TRUE);
	MpAlarmXHistory_0(Enable := TRUE);

	//TEST ALARM
	IF(TriggerAlarm)THEN
		MpAlarmXSet(MpLink := gAlarmXCoreLink, Name := 'AlarmTest');
		TriggerAlarm := FALSE;
	END_IF

END_PROGRAM

PROGRAM _EXIT

	MpAlarmXCoreObject(Enable := FALSE);
	MpAlarmXHistory_0(Enable := FALSE);

END_PROGRAM
```

### Program Logical/FileManager/FileManager (IEC)

#### Types.typ
```iecst
TYPE
	FileManagerUI : 	STRUCT
		MpFileManagerUI_0 : MpFileManagerUI;
		MpFileManagerUISetupType : MpFileManagerUISetupType;
		MpFileManagerUIConnectType : MpFileManagerUIConnectType;
		MpFileManagerUIFileListType : MpFileManagerUIFileListType;
		MpFileManagerUIFileType : MpFileManagerUIFileType;
		MpFileManagerUIItemType : MpFileManagerUIItemType;
	END_STRUCT;
	TableInfo : 	STRUCT
		Name : ARRAY[0..49]OF STRING[255];
		Size : ARRAY[0..49]OF UDINT;
		Type : ARRAY[0..49]OF MpFileManagerUIItemTypeEnum;
		LastModified : ARRAY[0..49]OF DATE_AND_TIME;
		NumberOfElements : USINT;
		SelectedRow : USINT;
	END_STRUCT;
	Auxiliary : 	STRUCT
		Two : STRING[160];
		One : STRING[160];
		Config1str : STRING[160];
		Config2str : STRING[160];
		Config3str : STRING[160];
		TableConfigurationStr : STRING[255];
		NumberOfElementsStr : STRING[80];
		errorNameExists : BOOL;
	END_STRUCT;
END_TYPE
```

#### Variables.var
```iecst
VAR
	cmd : FileManagerUI;
	iFile : USINT;
	tabInfo : TableInfo;
	aux : Auxiliary;
END_VAR
```

#### Main.st
```iecst
PROGRAM _INIT
	cmd.MpFileManagerUI_0.MpLink := ADR(gFileManagerUI);
	cmd.MpFileManagerUI_0.Enable := TRUE;

	cmd.MpFileManagerUI_0.UISetup := cmd.MpFileManagerUISetupType;
	cmd.MpFileManagerUI_0.UIConnect := ADR(cmd.MpFileManagerUIConnectType);

	(* define of device names *)
	cmd.MpFileManagerUIConnectType.DeviceList.DeviceNames[0] := 'UserPart';
	cmd.MpFileManagerUIConnectType.DeviceList.DeviceNames[1] := 'USB';

	cmd.MpFileManagerUI_0();
END_PROGRAM

PROGRAM _CYCLIC
	tabInfo.NumberOfElements := 0;
	aux.errorNameExists := 0;
	FOR iFile := 0 TO 49 BY 1 DO
		(* create arrays with file properties *)
		brsmemcpy(ADR(tabInfo.Name[iFile]), ADR(cmd.MpFileManagerUIConnectType.File.List.Items[iFile].Name), SIZEOF(tabInfo.Name[iFile]));
		brsmemcpy(ADR(tabInfo.Size[iFile]), ADR(cmd.MpFileManagerUIConnectType.File.List.Items[iFile].Size), SIZEOF(tabInfo.Size[iFile]));
		brsmemcpy(ADR(tabInfo.Type[iFile]), ADR(cmd.MpFileManagerUIConnectType.File.List.Items[iFile].ItemType), SIZEOF(tabInfo.Type[iFile]));
		brsmemcpy(ADR(tabInfo.LastModified[iFile]), ADR(cmd.MpFileManagerUIConnectType.File.List.Items[iFile].LastModified), SIZEOF(tabInfo.LastModified[iFile]));

		IF tabInfo.SelectedRow = iFile THEN
			cmd.MpFileManagerUIConnectType.File.List.Items[iFile].IsSelected := TRUE;
		END_IF
//
//		IF tabInfo.Name[iFile] = cmd.MpFileManagerUIConnectType.File.NewName AND (cmd.MpFileManagerUIConnectType THEN
//			aux.errorNameExists := 1;
//		END_IF

		(* dynamic change of the array size *)
		IF tabInfo.Type[iFile] <> mpFILE_ITEM_TYPE_NONE THEN
			tabInfo.NumberOfElements := tabInfo.NumberOfElements + 1;
		END_IF
	END_FOR;

	brsitoa(tabInfo.NumberOfElements, ADR(aux.NumberOfElementsStr));
	aux.TableConfigurationStr := '{"specRows": [ {"from":0, "to":';
	aux.One := ', "visible":true}, {"from":';
	aux.Two := ', "to":49, "visible":false}]}';
	brsstrcat(ADR(aux.TableConfigurationStr), ADR(aux.NumberOfElementsStr));
	brsstrcat(ADR(aux.TableConfigurationStr), ADR(aux.One));
	brsstrcat(ADR(aux.TableConfigurationStr), ADR(aux.NumberOfElementsStr));
	brsstrcat(ADR(aux.TableConfigurationStr), ADR(aux.Two));

	cmd.MpFileManagerUI_0();
END_PROGRAM

PROGRAM _EXIT
	(* Insert code here *)
	cmd.MpFileManagerUI_0.Enable := FALSE;
	cmd.MpFileManagerUI_0();
END_PROGRAM
```

### Types.typ - not listed in the package file held
```iecst
TYPE
	FileManagerUI : 	STRUCT
		MpFileManagerUI_0 : MpFileManagerUI;
		MpFileManagerUISetupType : MpFileManagerUISetupType;
		MpFileManagerUIConnectType : MpFileManagerUIConnectType;
		MpFileManagerUIFileListType : MpFileManagerUIFileListType;
		MpFileManagerUIFileType : MpFileManagerUIFileType;
		MpFileManagerUIItemType : MpFileManagerUIItemType;
	END_STRUCT;
	TableInfo : 	STRUCT
		Name : ARRAY[0..49]OF STRING[255];
		Size : ARRAY[0..49]OF UDINT;
		Type : ARRAY[0..49]OF MpFileManagerUIItemTypeEnum;
		LastModified : ARRAY[0..49]OF DATE_AND_TIME;
		NumberOfElements : USINT;
		SelectedRow : USINT;
	END_STRUCT;
	Auxiliary : 	STRUCT
		Two : STRING[160];
		One : STRING[160];
		Config1str : STRING[160];
		Config2str : STRING[160];
		Config3str : STRING[160];
		TableConfigurationStr : STRING[255];
		NumberOfElementsStr : STRING[80];
		NewNamePlus : USINT;
		NewNamePlusStr : STRING[80];
		NewNameTextOne : STRING[80];
		NewNameTextTwo : STRING[80];
		prevNewName : STRING[255];
		NumberOfElementsMinus : USINT;
		newNewName : STRING[255];
		btnSort : USINT;
		btnSortStr : STRING[80];
		fileName : STRING[260];
		fullFilePath : STRING[260];
		fileExtension3Chars : STRING[4];
		fileExtensionpdf : STRING[4] := '.pdf';
		fileExtensionPDF : STRING[4] := '.PDF';
		IsPDF : BOOL;
		fullFilePathWithFileDevice : STRING[260];
		SearchNewName : STRING[255];
		textStar : STRING[80] := '*';
	END_STRUCT;
END_TYPE
```
